LIN {X 0,Y 303.657,Z 547.41,A -85,B 0,C 180,E1 -15927.346,E2 -15927.346} C_VEL
LIN {X 0,Y 303.964,Z 546.683,A -85,B 0,C 180,E1 -15929.999,E2 -15929.999} C_VEL
LIN {X 0,Y 303.831,Z 546.451,A -85,B 0,C 180,E1 -15931.324,E2 -15931.324} C_VEL
LIN {X 0,Y 303.743,Z 545.822,A -85,B 0,C 180,E1 -15932.651,E2 -15932.651} C_VEL
LIN {X 0,Y 303.722,Z 544.801,A -85,B 0,C 180,E1 -15933.979,E2 -15933.979} C_VEL
LIN {X 0,Y 303.711,Z 542.811,A -85,B 0,C 180,E1 -15935.709,E2 -15935.709} C_VEL
LIN {X 0,Y 303.917,Z 539.098,A -85,B 0,C 180,E1 -15937.974,E2 -15937.974} C_VEL
LIN {X 0,Y 304.289,Z 534.652,A -85,B 0,C 180,E1 -15939.974,E2 -15939.974} C_VEL
LIN {X 0,Y 305.086,Z 527.886,A -85,B 0,C 180,E1 -15942.302,E2 -15942.302} C_VEL
LIN {X 0,Y 306.244,Z 520.516,A -85,B 0,C 180,E1 -15944.281,E2 -15944.281} C_VEL
LIN {X 0,Y 307.621,Z 511.711,A -85,B 0,C 180,E1 -15946.178,E2 -15946.178} C_VEL
LIN {X 0,Y 308.984,Z 501.769,A -85,B 0,C 180,E1 -15947.881,E2 -15947.881} C_VEL
LIN {X 0,Y 310.533,Z 491.16,A -85,B 0,C 180,E1 -15949.328,E2 -15949.328} C_VEL
LIN {X 0,Y 311.922,Z 480.889,A -85,B 0,C 180,E1 -15950.439,E2 -15950.439} C_VEL
LIN {X 0,Y 313.304,Z 468.561,A -85,B 0,C 180,E1 -15951.463,E2 -15951.463} C_VEL
LIN {X 0,Y 314.44,Z 455.612,A -85,B 0,C 180,E1 -15952.243,E2 -15952.243} C_VEL
LIN {X 0,Y 315.236,Z 443.183,A -85,B 0,C 180,E1 -15952.731,E2 -15952.731} C_VEL
LIN {X 0,Y 316.694,Z 379.006,A -85,B 0,C 180,E1 -15954.196,E2 -15954.196} C_VEL
LIN {X 0,Y 312.076,Z 344.443,A -85,B 0,C 180,E1 -15955.428,E2 -15955.428} C_VEL
LIN {X 0,Y 309.088,Z 325.843,A -85,B 0,C 180,E1 -15956.169,E2 -15956.169} C_VEL
LIN {X 0,Y 307.11,Z 315.452,A -85,B 0,C 180,E1 -15959.089,E2 -15959.089} C_VEL
LIN {X 0,Y 305.501,Z 307.431,A -85,B 0,C 180,E1 -15961.442,E2 -15961.442} C_VEL
LIN {X 0,Y 305.458,Z 307.433,A -85,B 0,C 180,E1 -15965.112,E2 -15965.112} C_VEL
LIN {X 0,Y 305.462,Z 307.434,A -85,B 0,C 180,E1 -15968.531,E2 -15968.531} C_VEL
LIN {X 0,Y 305.449,Z 307.432,A -85,B 0,C 180,E1 -15972.584,E2 -15972.584} C_VEL
LIN {X 0,Y 305.416,Z 307.436,A -85,B 0,C 180,E1 -15976.343,E2 -15976.343} C_VEL
LIN {X 0,Y 305.403,Z 307.44,A -85,B 0,C 180,E1 -15979.884,E2 -15979.884} C_VEL
LIN {X 0,Y 305.455,Z 307.437,A -85,B 0,C 180,E1 -15983.635,E2 -15983.635} C_VEL
LIN {X 0,Y 305.457,Z 307.433,A -85,B 0,C 180,E1 -15986.482,E2 -15986.482} C_VEL
LIN {X 0,Y 305.41,Z 307.44,A -85,B 0,C 180,E1 -15989.585,E2 -15989.585} C_VEL
LIN {X 0,Y 305.439,Z 307.436,A -85,B 0,C 180,E1 -15992.601,E2 -15992.601} C_VEL
LIN {X 0,Y 305.448,Z 307.436,A -85,B 0,C 180,E1 -15995.534,E2 -15995.534} C_VEL
LIN {X 0,Y 305.475,Z 307.427,A -85,B 0,C 180,E1 -15999.812,E2 -15999.812} C_VEL
LIN {X 0,Y 305.542,Z 307.416,A -85,B 0,C 180,E1 -16003.977,E2 -16003.977} C_VEL
LIN {X 0,Y 305.578,Z 307.417,A -85,B 0,C 180,E1 -16006.703,E2 -16006.703} C_VEL
LIN {X 0,Y 305.744,Z 307.395,A -85,B 0,C 180,E1 -16011.262,E2 -16011.262} C_VEL
LIN {X 0,Y 305.774,Z 307.379,A -85,B 0,C 180,E1 -16013.401,E2 -16013.401} C_VEL
LIN {X 0,Y 305.847,Z 307.383,A -85,B 0,C 180,E1 -16017.366,E2 -16017.366} C_VEL
LIN {X 0,Y 305.903,Z 307.377,A -85,B 0,C 180,E1 -16020,E2 -16020} C_VEL
LIN {X 0,Y 305.842,Z 307.385,A -85,B 0,C 180,E1 -16022.634,E2 -16022.634} C_VEL
LIN {X 0,Y 305.775,Z 307.395,A -85,B 0,C 180,E1 -16026.599,E2 -16026.599} C_VEL
LIN {X 0,Y 305.686,Z 307.404,A -85,B 0,C 180,E1 -16029.261,E2 -16029.261} C_VEL
LIN {X 0,Y 305.578,Z 307.42,A -85,B 0,C 180,E1 -16033.297,E2 -16033.297} C_VEL
LIN {X 0,Y 305.543,Z 307.418,A -85,B 0,C 180,E1 -16036.023,E2 -16036.023} C_VEL
LIN {X 0,Y 305.534,Z 307.424,A -85,B 0,C 180,E1 -16039.427,E2 -16039.427} C_VEL
LIN {X 0,Y 305.479,Z 307.43,A -85,B 0,C 180,E1 -16043.04,E2 -16043.04} C_VEL
LIN {X 0,Y 305.47,Z 307.428,A -85,B 0,C 180,E1 -16046.201,E2 -16046.201} C_VEL
LIN {X 0,Y 305.456,Z 307.435,A -85,B 0,C 180,E1 -16049.04,E2 -16049.04} C_VEL
LIN {X 0,Y 305.43,Z 307.432,A -85,B 0,C 180,E1 -16051.954,E2 -16051.954} C_VEL
LIN {X 0,Y 305.456,Z 307.435,A -85,B 0,C 180,E1 -16055.114,E2 -16055.114} C_VEL
LIN {X 0,Y 305.443,Z 307.435,A -85,B 0,C 180,E1 -16058.53,E2 -16058.53} C_VEL
LIN {X 0,Y 305.449,Z 307.434,A -85,B 0,C 180,E1 -16062.587,E2 -16062.587} C_VEL
LIN {X 0,Y 305.421,Z 307.441,A -85,B 0,C 180,E1 -16066.346,E2 -16066.346} C_VEL
LIN {X 0,Y 305.454,Z 307.436,A -85,B 0,C 180,E1 -16069.894,E2 -16069.894} C_VEL
LIN {X 0,Y 305.478,Z 307.424,A -85,B 0,C 180,E1 -16073.633,E2 -16073.633} C_VEL
LIN {X 0,Y 305.462,Z 307.434,A -85,B 0,C 180,E1 -16076.485,E2 -16076.485} C_VEL
LIN {X 0,Y 305.455,Z 307.433,A -85,B 0,C 180,E1 -16079.592,E2 -16079.592} C_VEL
LIN {X 0,Y 305.526,Z 307.425,A -85,B 0,C 180,E1 -16083.469,E2 -16083.469} C_VEL
LIN {X 0,Y 306.651,Z 310.421,A -85,B 0,C 180,E1 -16083.666,E2 -16083.666} C_VEL
LIN {X 0,Y 315.433,Z 329.159,A -85,B 0,C 180,E1 -16084.926,E2 -16084.926} C_VEL
LIN {X 0,Y 318.099,Z 335.429,A -85,B 0,C 180,E1 -16085.306,E2 -16085.306} C_VEL
LIN {X 0,Y 317.199,Z 379.67,A -85,B 0,C 180,E1 -16086.313,E2 -16086.313} C_VEL
LIN {X 0,Y 316.238,Z 417.455,A -85,B 0,C 180,E1 -16087.201,E2 -16087.201} C_VEL
LIN {X 0,Y 315.569,Z 430.397,A -85,B 0,C 180,E1 -16087.754,E2 -16087.754} C_VEL
LIN {X 0,Y 314.521,Z 443.873,A -85,B 0,C 180,E1 -16088.624,E2 -16088.624} C_VEL
LIN {X 0,Y 313.322,Z 455.582,A -85,B 0,C 180,E1 -16089.656,E2 -16089.656} C_VEL
LIN {X 0,Y 311.905,Z 466.753,A -85,B 0,C 180,E1 -16090.932,E2 -16090.932} C_VEL
LIN {X 0,Y 310.754,Z 476.06,A -85,B 0,C 180,E1 -16092.267,E2 -16092.267} C_VEL
LIN {X 0,Y 309.297,Z 485.106,A -85,B 0,C 180,E1 -16093.84,E2 -16093.84} C_VEL
LIN {X 0,Y 307.998,Z 492.729,A -85,B 0,C 180,E1 -16095.465,E2 -16095.465} C_VEL
LIN {X 0,Y 306.779,Z 500.157,A -85,B 0,C 180,E1 -16097.431,E2 -16097.431} C_VEL
LIN {X 0,Y 305.743,Z 506.122,A -85,B 0,C 180,E1 -16099.405,E2 -16099.405} C_VEL
LIN {X 0,Y 304.994,Z 510.833,A -85,B 0,C 180,E1 -16101.387,E2 -16101.387} C_VEL
LIN {X 0,Y 304.481,Z 514.431,A -85,B 0,C 180,E1 -16103.374,E2 -16103.374} C_VEL
LIN {X 0,Y 304.244,Z 516.283,A -85,B 0,C 180,E1 -16104.7,E2 -16104.7} C_VEL
LIN {X 0,Y 304.001,Z 517.699,A -85,B 0,C 180,E1 -16106.024,E2 -16106.024} C_VEL
LIN {X 0,Y 303.771,Z 519.302,A -85,B 0,C 180,E1 -16108.676,E2 -16108.676} C_VEL
LIN {X 0,Y 303.767,Z 519.534,A -85,B 0,C 180,E1 -16110.001,E2 -16110.001} C_VEL
LIN {X 0,Y 303.771,Z 519.341,A -85,B 0,C 180,E1 -16111.327,E2 -16111.327} C_VEL
LIN {X 0,Y 303.998,Z 517.791,A -85,B 0,C 180,E1 -16113.978,E2 -16113.978} C_VEL
LIN {X 0,Y 304.24,Z 516.425,A -85,B 0,C 180,E1 -16115.303,E2 -16115.303} C_VEL
LIN {X 0,Y 304.624,Z 513.67,A -85,B 0,C 180,E1 -16117.225,E2 -16117.225} C_VEL
LIN {X 0,Y 305.149,Z 509.667,A -85,B 0,C 180,E1 -16119.279,E2 -16119.279} C_VEL
LIN {X 0,Y 306.027,Z 504.616,A -85,B 0,C 180,E1 -16121.258,E2 -16121.258} C_VEL
LIN {X 0,Y 307.119,Z 498.247,A -85,B 0,C 180,E1 -16123.23,E2 -16123.23} C_VEL
LIN {X 0,Y 308.437,Z 490.319,A -85,B 0,C 180,E1 -16125.192,E2 -16125.192} C_VEL
LIN {X 0,Y 309.862,Z 482.199,A -85,B 0,C 180,E1 -16126.81,E2 -16126.81} C_VEL
LIN {X 0,Y 311.249,Z 472.224,A -85,B 0,C 180,E1 -16128.43,E2 -16128.43} C_VEL
LIN {X 0,Y 312.689,Z 461.004,A -85,B 0,C 180,E1 -16129.875,E2 -16129.875} C_VEL
LIN {X 0,Y 313.976,Z 449.96,A -85,B 0,C 180,E1 -16130.987,E2 -16130.987} C_VEL
LIN {X 0,Y 315.116,Z 437.46,A -85,B 0,C 180,E1 -16131.937,E2 -16131.937} C_VEL
LIN {X 0,Y 315.979,Z 424.357,A -85,B 0,C 180,E1 -16132.649,E2 -16132.649} C_VEL
LIN {X 0,Y 316.472,Z 411.322,A -85,B 0,C 180,E1 -16133.086,E2 -16133.086} C_VEL
LIN {X 0,Y 318.254,Z 335.871,A -85,B 0,C 180,E1 -16134.785,E2 -16134.785} C_VEL
LIN {X 0,Y 310.377,Z 318.013,A -85,B 0,C 180,E1 -16135.916,E2 -16135.916} C_VEL
LIN {X 0,Y 305.665,Z 308.157,A -85,B 0,C 180,E1 -16136.604,E2 -16136.604} C_VEL
LIN {X 0,Y 305.53,Z 307.424,A -85,B 0,C 180,E1 -16136.661,E2 -16136.661} C_VEL
LIN {X 0,Y 305.468,Z 307.433,A -85,B 0,C 180,E1 -16140.41,E2 -16140.41} C_VEL
LIN {X 0,Y 305.47,Z 307.434,A -85,B 0,C 180,E1 -16144.079,E2 -16144.079} C_VEL
LIN {X 0,Y 305.501,Z 307.427,A -85,B 0,C 180,E1 -16146.737,E2 -16146.737} C_VEL
LIN {X 0,Y 305.459,Z 307.435,A -85,B 0,C 180,E1 -16150.614,E2 -16150.614} C_VEL
LIN {X 0,Y 305.451,Z 307.432,A -85,B 0,C 180,E1 -16153.652,E2 -16153.652} C_VEL
LIN {X 0,Y 305.448,Z 307.421,A -85,B 0,C 180,E1 -16156.346,E2 -16156.346} C_VEL
LIN {X 0,Y 304.825,Z 307.507,A -85,B 0,C 180,E1 -16157.445,E2 -16157.445} C_VEL
LIN {X 0,Y 301.944,Z 307.873,A -85,B 0,C 180,E1 -16159.235,E2 -16159.235} C_VEL
LIN {X 0,Y 299.493,Z 308.179,A -85,B 0,C 180,E1 -16160.687,E2 -16160.687} C_VEL
LIN {X 0,Y 298.473,Z 308.303,A -85,B 0,C 180,E1 -16161.812,E2 -16161.812} C_VEL
LIN {X 0,Y 298.41,Z 308.31,A -85,B 0,C 180,E1 -16162.194,E2 -16162.194} C_VEL
LIN {X 0,Y 298.414,Z 308.312,A -85,B 0,C 180,E1 -16165.582,E2 -16165.582} C_VEL
LIN {X 0,Y 298.397,Z 308.311,A -85,B 0,C 180,E1 -16168.791,E2 -16168.791} C_VEL
LIN {X 0,Y 298.463,Z 308.305,A -85,B 0,C 180,E1 -16171.904,E2 -16171.904} C_VEL
LIN {X 0,Y 298.52,Z 308.295,A -85,B 0,C 180,E1 -16176.039,E2 -16176.039} C_VEL
LIN {X 0,Y 298.545,Z 308.359,A -85,B 0,C 180,E1 -16176.41,E2 -16176.41} C_VEL
LIN {X 0,Y 298.71,Z 309.327,A -85,B 0,C 180,E1 -16176.684,E2 -16176.684} C_VEL
LIN {X 0,Y 304.792,Z 332.568,A -85,B 0,C 180,E1 -16177.782,E2 -16177.782} C_VEL
LIN {X 0,Y 305.454,Z 337.875,A -85,B 0,C 180,E1 -16177.999,E2 -16177.999} C_VEL
LIN {X 0,Y 302.641,Z 418.79,A -85,B 0,C 180,E1 -16180.852,E2 -16180.852} C_VEL
LIN {X 0,Y 302.093,Z 432.467,A -85,B 0,C 180,E1 -16181.607,E2 -16181.607} C_VEL
LIN {X 0,Y 301.327,Z 444.568,A -85,B 0,C 180,E1 -16182.526,E2 -16182.526} C_VEL
LIN {X 0,Y 300.57,Z 456.641,A -85,B 0,C 180,E1 -16183.705,E2 -16183.705} C_VEL
LIN {X 0,Y 300.027,Z 465.153,A -85,B 0,C 180,E1 -16184.72,E2 -16184.72} C_VEL
LIN {X 0,Y 299.157,Z 475.798,A -85,B 0,C 180,E1 -16186.239,E2 -16186.239} C_VEL
LIN {X 0,Y 298.337,Z 486.282,A -85,B 0,C 180,E1 -16188.104,E2 -16188.104} C_VEL
LIN {X 0,Y 297.698,Z 495.551,A -85,B 0,C 180,E1 -16190.145,E2 -16190.145} C_VEL
LIN {X 0,Y 297.211,Z 502.937,A -85,B 0,C 180,E1 -16192.185,E2 -16192.185} C_VEL
LIN {X 0,Y 296.851,Z 509.748,A -85,B 0,C 180,E1 -16194.566,E2 -16194.566} C_VEL
LIN {X 0,Y 296.772,Z 514.18,A -85,B 0,C 180,E1 -16196.606,E2 -16196.606} C_VEL
LIN {X 0,Y 296.617,Z 517.475,A -85,B 0,C 180,E1 -16198.642,E2 -16198.642} C_VEL
LIN {X 0,Y 296.63,Z 519.071,A -85,B 0,C 180,E1 -16200,E2 -16200} C_VEL
LIN {X 0,Y 296.736,Z 520.242,A -85,B 0,C 180,E1 -16201.357,E2 -16201.357} C_VEL
LIN {X 0,Y 296.924,Z 520.999,A -85,B 0,C 180,E1 -16202.713,E2 -16202.713} C_VEL
LIN {X 0,Y 297.161,Z 521.297,A -85,B 0,C 180,E1 -16204.069,E2 -16204.069} C_VEL
LIN {X 0,Y 297.378,Z 521.168,A -85,B 0,C 180,E1 -16205.424,E2 -16205.424} C_VEL
LIN {X 0,Y 297.751,Z 520.634,A -85,B 0,C 180,E1 -16206.778,E2 -16206.778} C_VEL
LIN {X 0,Y 298.641,Z 519.069,A -85,B 0,C 180,E1 -16208.731,E2 -16208.731} C_VEL
LIN {X 0,Y 300.157,Z 515.318,A -85,B 0,C 180,E1 -16211.48,E2 -16211.48} C_VEL
LIN {X 0,Y 301.698,Z 511.3,A -85,B 0,C 180,E1 -16213.471,E2 -16213.471} C_VEL
LIN {X 0,Y 303.4,Z 506.16,A -85,B 0,C 180,E1 -16215.449,E2 -16215.449} C_VEL
LIN {X 0,Y 305.88,Z 498.522,A -85,B 0,C 180,E1 -16217.724,E2 -16217.724} C_VEL
LIN {X 0,Y 308.402,Z 490.221,A -85,B 0,C 180,E1 -16219.641,E2 -16219.641} C_VEL
LIN {X 0,Y 311.29,Z 479.988,A -85,B 0,C 180,E1 -16221.523,E2 -16221.523} C_VEL
LIN {X 0,Y 314.004,Z 469.151,A -85,B 0,C 180,E1 -16223.104,E2 -16223.104} C_VEL
LIN {X 0,Y 316.565,Z 457.559,A -85,B 0,C 180,E1 -16224.46,E2 -16224.46} C_VEL
LIN {X 0,Y 318.939,Z 444.809,A -85,B 0,C 180,E1 -16225.623,E2 -16225.623} C_VEL
LIN {X 0,Y 320.899,Z 432.294,A -85,B 0,C 180,E1 -16226.502,E2 -16226.502} C_VEL
LIN {X 0,Y 322.631,Z 418.016,A -85,B 0,C 180,E1 -16227.223,E2 -16227.223} C_VEL
LIN {X 0,Y 329.241,Z 360.312,A -85,B 0,C 180,E1 -16229.538,E2 -16229.538} C_VEL
LIN {X 0,Y 325.595,Z 352.92,A -85,B 0,C 180,E1 -16231.008,E2 -16231.008} C_VEL
LIN {X 0,Y 322.312,Z 347.353,A -85,B 0,C 180,E1 -16232.44,E2 -16232.44} C_VEL
LIN {X 0,Y 318.784,Z 341.964,A -85,B 0,C 180,E1 -16234.186,E2 -16234.186} C_VEL
LIN {X 0,Y 315.89,Z 337.946,A -85,B 0,C 180,E1 -16235.88,E2 -16235.88} C_VEL
LIN {X 0,Y 312.534,Z 333.726,A -85,B 0,C 180,E1 -16238.417,E2 -16238.417} C_VEL
LIN {X 0,Y 309.76,Z 331.31,A -85,B 0,C 180,E1 -16241.74,E2 -16241.74} C_VEL
LIN {X 0,Y 309.236,Z 330.576,A -85,B 0,C 180,E1 -16243.341,E2 -16243.341} C_VEL
LIN {X 0,Y 309.074,Z 331.036,A -85,B 0,C 180,E1 -16245.474,E2 -16245.474} C_VEL
LIN {X 0,Y 309.758,Z 332.653,A -85,B 0,C 180,E1 -16247.724,E2 -16247.724} C_VEL
LIN {X 0,Y 311.676,Z 336.685,A -85,B 0,C 180,E1 -16250.482,E2 -16250.482} C_VEL
LIN {X 0,Y 314.583,Z 341.177,A -85,B 0,C 180,E1 -16252.879,E2 -16252.879} C_VEL
LIN {X 0,Y 318.33,Z 348.268,A -85,B 0,C 180,E1 -16255.268,E2 -16255.268} C_VEL
LIN {X 0,Y 321.308,Z 354.437,A -85,B 0,C 180,E1 -16256.849,E2 -16256.849} C_VEL
LIN {X 0,Y 323.815,Z 360.163,A -85,B 0,C 180,E1 -16258.057,E2 -16258.057} C_VEL
LIN {X 0,Y 324.995,Z 363.139,A -85,B 0,C 180,E1 -16258.6,E2 -16258.6} C_VEL
LIN {X 0,Y 326.341,Z 374.009,A -85,B 0,C 180,E1 -16259.718,E2 -16259.718} C_VEL
LIN {X 0,Y 327.059,Z 384.878,A -85,B 0,C 180,E1 -16260.612,E2 -16260.612} C_VEL
LIN {X 0,Y 321.516,Z 436.451,A -85,B 0,C 180,E1 -16262.674,E2 -16262.674} C_VEL
LIN {X 0,Y 319.542,Z 451.172,A -85,B 0,C 180,E1 -16263.375,E2 -16263.375} C_VEL
LIN {X 0,Y 316.795,Z 466.219,A -85,B 0,C 180,E1 -16264.366,E2 -16264.366} C_VEL
LIN {X 0,Y 314.332,Z 477.863,A -85,B 0,C 180,E1 -16265.389,E2 -16265.389} C_VEL
LIN {X 0,Y 311.455,Z 490.024,A -85,B 0,C 180,E1 -16266.74,E2 -16266.74} C_VEL
LIN {X 0,Y 308.656,Z 501.054,A -85,B 0,C 180,E1 -16268.283,E2 -16268.283} C_VEL
LIN {X 0,Y 306.177,Z 510.183,A -85,B 0,C 180,E1 -16269.859,E2 -16269.859} C_VEL
LIN {X 0,Y 303.687,Z 518.633,A -85,B 0,C 180,E1 -16271.619,E2 -16271.619} C_VEL
LIN {X 0,Y 301.519,Z 526.799,A -85,B 0,C 180,E1 -16273.756,E2 -16273.756} C_VEL
LIN {X 0,Y 299.822,Z 532.872,A -85,B 0,C 180,E1 -16275.75,E2 -16275.75} C_VEL
LIN {X 0,Y 298.46,Z 537.761,A -85,B 0,C 180,E1 -16277.763,E2 -16277.763} C_VEL
LIN {X 0,Y 297.5,Z 541.558,A -85,B 0,C 180,E1 -16279.793,E2 -16279.793} C_VEL
LIN {X 0,Y 296.894,Z 544.333,A -85,B 0,C 180,E1 -16281.833,E2 -16281.833} C_VEL
LIN {X 0,Y 296.581,Z 546.422,A -85,B 0,C 180,E1 -16284.422,E2 -16284.422} C_VEL
LIN {X 0,Y 296.572,Z 546.955,A -85,B 0,C 180,E1 -16285.922,E2 -16285.922} C_VEL
LIN {X 0,Y 296.58,Z 546.981,A -85,B 0,C 180,E1 -16287.282,E2 -16287.282} C_VEL
LIN {X 0,Y 296.866,Z 546.366,A -85,B 0,C 180,E1 -16289.999,E2 -16289.999} C_VEL
LIN {X 0,Y 296.735,Z 546.133,A -85,B 0,C 180,E1 -16291.356,E2 -16291.356} C_VEL
LIN {X 0,Y 296.661,Z 545.505,A -85,B 0,C 180,E1 -16292.714,E2 -16292.714} C_VEL
LIN {X 0,Y 296.631,Z 544.483,A -85,B 0,C 180,E1 -16294.075,E2 -16294.075} C_VEL
LIN {X 0,Y 296.623,Z 542.739,A -85,B 0,C 180,E1 -16295.659,E2 -16295.659} C_VEL
LIN {X 0,Y 296.852,Z 538.78,A -85,B 0,C 180,E1 -16298.165,E2 -16298.165} C_VEL
LIN {X 0,Y 297.251,Z 534.333,A -85,B 0,C 180,E1 -16300.213,E2 -16300.213} C_VEL
LIN {X 0,Y 297.94,Z 528.667,A -85,B 0,C 180,E1 -16302.256,E2 -16302.256} C_VEL
LIN {X 0,Y 299.15,Z 521.553,A -85,B 0,C 180,E1 -16304.28,E2 -16304.28} C_VEL
LIN {X 0,Y 300.572,Z 512.685,A -85,B 0,C 180,E1 -16306.294,E2 -16306.294} C_VEL
LIN {X 0,Y 301.899,Z 503.565,A -85,B 0,C 180,E1 -16307.964,E2 -16307.964} C_VEL
LIN {X 0,Y 303.457,Z 493.414,A -85,B 0,C 180,E1 -16309.445,E2 -16309.445} C_VEL
LIN {X 0,Y 305.071,Z 482.154,A -85,B 0,C 180,E1 -16310.743,E2 -16310.743} C_VEL
LIN {X 0,Y 306.465,Z 470.457,A -85,B 0,C 180,E1 -16311.789,E2 -16311.789} C_VEL
LIN {X 0,Y 307.691,Z 457.555,A -85,B 0,C 180,E1 -16312.625,E2 -16312.625} C_VEL
LIN {X 0,Y 308.64,Z 444.389,A -85,B 0,C 180,E1 -16313.193,E2 -16313.193} C_VEL
LIN {X 0,Y 309.973,Z 393.218,A -85,B 0,C 180,E1 -16314.397,E2 -16314.397} C_VEL
LIN {X 0,Y 310.199,Z 379.909,A -85,B 0,C 180,E1 -16314.708,E2 -16314.708} C_VEL
LIN {X 0,Y 305.808,Z 346.318,A -85,B 0,C 180,E1 -16315.934,E2 -16315.934} C_VEL
LIN {X 0,Y 302.785,Z 328.078,A -85,B 0,C 180,E1 -16316.681,E2 -16316.681} C_VEL
LIN {X 0,Y 301.693,Z 324.321,A -85,B 0,C 180,E1 -16316.9,E2 -16316.9} C_VEL
LIN {X 0,Y 298.974,Z 310.991,A -85,B 0,C 180,E1 -16320.779,E2 -16320.779} C_VEL
LIN {X 0,Y 298.462,Z 308.308,A -85,B 0,C 180,E1 -16321.635,E2 -16321.635} C_VEL
LIN {X 0,Y 298.415,Z 308.314,A -85,B 0,C 180,E1 -16326.068,E2 -16326.068} C_VEL
LIN {X 0,Y 298.404,Z 308.313,A -85,B 0,C 180,E1 -16329.485,E2 -16329.485} C_VEL
LIN {X 0,Y 298.394,Z 308.311,A -85,B 0,C 180,E1 -16333.102,E2 -16333.102} C_VEL
LIN {X 0,Y 298.365,Z 308.312,A -85,B 0,C 180,E1 -16336.914,E2 -16336.914} C_VEL
LIN {X 0,Y 298.344,Z 308.314,A -85,B 0,C 180,E1 -16341.018,E2 -16341.018} C_VEL
LIN {X 0,Y 298.397,Z 308.312,A -85,B 0,C 180,E1 -16343.927,E2 -16343.927} C_VEL
LIN {X 0,Y 298.385,Z 308.315,A -85,B 0,C 180,E1 -16347.198,E2 -16347.198} C_VEL
LIN {X 0,Y 298.36,Z 308.316,A -85,B 0,C 180,E1 -16350.636,E2 -16350.636} C_VEL
LIN {X 0,Y 298.413,Z 308.308,A -85,B 0,C 180,E1 -16354.917,E2 -16354.917} C_VEL
LIN {X 0,Y 298.393,Z 308.315,A -85,B 0,C 180,E1 -16357.862,E2 -16357.862} C_VEL
LIN {X 0,Y 298.456,Z 308.299,A -85,B 0,C 180,E1 -16360.751,E2 -16360.751} C_VEL
LIN {X 0,Y 298.578,Z 308.283,A -85,B 0,C 180,E1 -16364.994,E2 -16364.994} C_VEL
LIN {X 0,Y 298.574,Z 308.294,A -85,B 0,C 180,E1 -16369.146,E2 -16369.146} C_VEL
LIN {X 0,Y 298.687,Z 308.268,A -85,B 0,C 180,E1 -16371.884,E2 -16371.884} C_VEL
LIN {X 0,Y 298.619,Z 308.264,A -85,B 0,C 180,E1 -16374.598,E2 -16374.598} C_VEL
LIN {X 0,Y 298.894,Z 308.249,A -85,B 0,C 180,E1 -16378.653,E2 -16378.653} C_VEL
LIN {X 0,Y 298.903,Z 308.251,A -85,B 0,C 180,E1 -16381.347,E2 -16381.347} C_VEL
LIN {X 0,Y 298.724,Z 308.275,A -85,B 0,C 180,E1 -16386.756,E2 -16386.756} C_VEL
LIN {X 0,Y 298.617,Z 308.282,A -85,B 0,C 180,E1 -16389.483,E2 -16389.483} C_VEL
LIN {X 0,Y 298.537,Z 308.295,A -85,B 0,C 180,E1 -16393.616,E2 -16393.616} C_VEL
LIN {X 0,Y 298.478,Z 308.299,A -85,B 0,C 180,E1 -16396.413,E2 -16396.413} C_VEL
LIN {X 0,Y 298.475,Z 308.302,A -85,B 0,C 180,E1 -16399.64,E2 -16399.64} C_VEL
LIN {X 0,Y 298.417,Z 308.306,A -85,B 0,C 180,E1 -16403.601,E2 -16403.601} C_VEL
LIN {X 0,Y 298.409,Z 308.31,A -85,B 0,C 180,E1 -16406.582,E2 -16406.582} C_VEL
LIN {X 0,Y 298.393,Z 308.313,A -85,B 0,C 180,E1 -16409.644,E2 -16409.644} C_VEL
LIN {X 0,Y 298.386,Z 308.313,A -85,B 0,C 180,E1 -16412.802,E2 -16412.802} C_VEL
LIN {X 0,Y 298.44,Z 308.306,A -85,B 0,C 180,E1 -16416.809,E2 -16416.809} C_VEL
LIN {X 0,Y 298.381,Z 308.315,A -85,B 0,C 180,E1 -16421.089,E2 -16421.089} C_VEL
LIN {X 0,Y 298.393,Z 308.311,A -85,B 0,C 180,E1 -16423.105,E2 -16423.105} C_VEL
LIN {X 0,Y 298.398,Z 308.311,A -85,B 0,C 180,E1 -16426.922,E2 -16426.922} C_VEL
LIN {X 0,Y 298.411,Z 308.308,A -85,B 0,C 180,E1 -16431.005,E2 -16431.005} C_VEL
LIN {X 0,Y 298.415,Z 308.305,A -85,B 0,C 180,E1 -16433.932,E2 -16433.932} C_VEL
LIN {X 0,Y 298.39,Z 308.309,A -85,B 0,C 180,E1 -16437.985,E2 -16437.985} C_VEL
LIN {X 0,Y 298.457,Z 308.307,A -85,B 0,C 180,E1 -16441.905,E2 -16441.905} C_VEL
LIN {X 0,Y 298.479,Z 308.303,A -85,B 0,C 180,E1 -16442.811,E2 -16442.811} C_VEL
LIN {X 0,Y 299.494,Z 311.154,A -85,B 0,C 180,E1 -16442.999,E2 -16442.999} C_VEL
LIN {X 0,Y 307.474,Z 327.59,A -85,B 0,C 180,E1 -16444.183,E2 -16444.183} C_VEL
LIN {X 0,Y 311.683,Z 337.348,A -85,B 0,C 180,E1 -16444.805,E2 -16444.805} C_VEL
LIN {X 0,Y 309.917,Z 412.201,A -85,B 0,C 180,E1 -16446.532,E2 -16446.532} C_VEL
LIN {X 0,Y 309.396,Z 424.986,A -85,B 0,C 180,E1 -16446.977,E2 -16446.977} C_VEL
LIN {X 0,Y 308.563,Z 437.395,A -85,B 0,C 180,E1 -16447.663,E2 -16447.663} C_VEL
LIN {X 0,Y 307.42,Z 449.046,A -85,B 0,C 180,E1 -16448.546,E2 -16448.546} C_VEL
LIN {X 0,Y 306.108,Z 460.416,A -85,B 0,C 180,E1 -16449.682,E2 -16449.682} C_VEL
LIN {X 0,Y 304.604,Z 471.8,A -85,B 0,C 180,E1 -16451.156,E2 -16451.156} C_VEL
LIN {X 0,Y 303.114,Z 481.944,A -85,B 0,C 180,E1 -16452.807,E2 -16452.807} C_VEL
LIN {X 0,Y 301.637,Z 490.16,A -85,B 0,C 180,E1 -16454.46,E2 -16454.46} C_VEL
LIN {X 0,Y 300.276,Z 498.161,A -85,B 0,C 180,E1 -16456.466,E2 -16456.466} C_VEL
LIN {X 0,Y 299.123,Z 504.606,A -85,B 0,C 180,E1 -16458.481,E2 -16458.481} C_VEL
LIN {X 0,Y 298.209,Z 509.728,A -85,B 0,C 180,E1 -16460.506,E2 -16460.506} C_VEL
LIN {X 0,Y 297.56,Z 514.026,A -85,B 0,C 180,E1 -16462.744,E2 -16462.744} C_VEL
LIN {X 0,Y 297.178,Z 516.6,A -85,B 0,C 180,E1 -16464.573,E2 -16464.573} C_VEL
LIN {X 0,Y 296.941,Z 518.015,A -85,B 0,C 180,E1 -16465.93,E2 -16465.93} C_VEL
LIN {X 0,Y 296.684,Z 519.619,A -85,B 0,C 180,E1 -16468.644,E2 -16468.644} C_VEL
LIN {X 0,Y 296.675,Z 519.851,A -85,B 0,C 180,E1 -16470.001,E2 -16470.001} C_VEL
LIN {X 0,Y 296.684,Z 519.658,A -85,B 0,C 180,E1 -16471.359,E2 -16471.359} C_VEL
LIN {X 0,Y 296.938,Z 518.106,A -85,B 0,C 180,E1 -16474.073,E2 -16474.073} C_VEL
LIN {X 0,Y 297.174,Z 516.741,A -85,B 0,C 180,E1 -16475.43,E2 -16475.43} C_VEL
LIN {X 0,Y 297.542,Z 514.242,A -85,B 0,C 180,E1 -16477.229,E2 -16477.229} C_VEL
LIN {X 0,Y 298.132,Z 509.982,A -85,B 0,C 180,E1 -16479.499,E2 -16479.499} C_VEL
LIN {X 0,Y 299.074,Z 504.929,A -85,B 0,C 180,E1 -16481.523,E2 -16481.523} C_VEL
LIN {X 0,Y 300.229,Z 498.558,A -85,B 0,C 180,E1 -16483.539,E2 -16483.539} C_VEL
LIN {X 0,Y 301.595,Z 490.629,A -85,B 0,C 180,E1 -16485.545,E2 -16485.545} C_VEL
LIN {X 0,Y 303.068,Z 482.507,A -85,B 0,C 180,E1 -16487.199,E2 -16487.199} C_VEL
LIN {X 0,Y 304.525,Z 472.528,A -85,B 0,C 180,E1 -16488.852,E2 -16488.852} C_VEL
LIN {X 0,Y 306.038,Z 461.303,A -85,B 0,C 180,E1 -16490.326,E2 -16490.326} C_VEL
LIN {X 0,Y 307.389,Z 450.25,A -85,B 0,C 180,E1 -16491.459,E2 -16491.459} C_VEL
LIN {X 0,Y 308.549,Z 437.738,A -85,B 0,C 180,E1 -16492.429,E2 -16492.429} C_VEL
LIN {X 0,Y 309.467,Z 424.613,A -85,B 0,C 180,E1 -16493.153,E2 -16493.153} C_VEL
LIN {X 0,Y 309.978,Z 411.518,A -85,B 0,C 180,E1 -16493.599,E2 -16493.599} C_VEL
LIN {X 0,Y 311.805,Z 337.588,A -85,B 0,C 180,E1 -16495.295,E2 -16495.295} C_VEL
LIN {X 0,Y 303.699,Z 319.52,A -85,B 0,C 180,E1 -16496.495,E2 -16496.495} C_VEL
LIN {X 0,Y 298.704,Z 309.41,A -85,B 0,C 180,E1 -16497.246,E2 -16497.246} C_VEL
LIN {X 0,Y 298.483,Z 308.303,A -85,B 0,C 180,E1 -16497.337,E2 -16497.337} C_VEL
LIN {X 0,Y 298.401,Z 308.315,A -85,B 0,C 180,E1 -16501.21,E2 -16501.21} C_VEL
LIN {X 0,Y 298.433,Z 308.309,A -85,B 0,C 180,E1 -16504.488,E2 -16504.488} C_VEL
LIN {X 0,Y 298.437,Z 308.314,A -85,B 0,C 180,E1 -16507.756,E2 -16507.756} C_VEL
LIN {X 0,Y 298.418,Z 308.316,A -85,B 0,C 180,E1 -16511.257,E2 -16511.257} C_VEL
LIN {X 0,Y 298.394,Z 308.302,A -85,B 0,C 180,E1 -16515.042,E2 -16515.042} C_VEL
LIN {X 0,Y 298.393,Z 308.312,A -85,B 0,C 180,E1 -16518.913,E2 -16518.913} C_VEL
LIN {X 0,Y 298.41,Z 308.31,A -85,B 0,C 180,E1 -16522.194,E2 -16522.194} C_VEL
LIN {X 0,Y 297.805,Z 308.388,A -85,B 0,C 180,E1 -16523.32,E2 -16523.32} C_VEL
LIN {X 0,Y 294.995,Z 308.742,A -85,B 0,C 180,E1 -16525.155,E2 -16525.155} C_VEL
LIN {X 0,Y 292.552,Z 309.045,A -85,B 0,C 180,E1 -16526.643,E2 -16526.643} C_VEL
LIN {X 0,Y 291.464,Z 309.175,A -85,B 0,C 180,E1 -16527.796,E2 -16527.796} C_VEL
LIN {X 0,Y 291.356,Z 309.186,A -85,B 0,C 180,E1 -16528.187,E2 -16528.187} C_VEL
LIN {X 0,Y 291.383,Z 309.19,A -85,B 0,C 180,E1 -16531.158,E2 -16531.158} C_VEL
LIN {X 0,Y 291.424,Z 309.182,A -85,B 0,C 180,E1 -16534.272,E2 -16534.272} C_VEL
LIN {X 0,Y 291.506,Z 309.237,A -85,B 0,C 180,E1 -16536.296,E2 -16536.296} C_VEL
LIN {X 0,Y 291.676,Z 310.186,A -85,B 0,C 180,E1 -16536.419,E2 -16536.419} C_VEL
LIN {X 0,Y 297.96,Z 334.104,A -85,B 0,C 180,E1 -16537.575,E2 -16537.575} C_VEL
LIN {X 0,Y 298.474,Z 338.793,A -85,B 0,C 180,E1 -16537.769,E2 -16537.769} C_VEL
LIN {X 0,Y 295.601,Z 418.979,A -85,B 0,C 180,E1 -16540.693,E2 -16540.693} C_VEL
LIN {X 0,Y 295.063,Z 431.929,A -85,B 0,C 180,E1 -16541.423,E2 -16541.423} C_VEL
LIN {X 0,Y 294.265,Z 444.694,A -85,B 0,C 180,E1 -16542.406,E2 -16542.406} C_VEL
LIN {X 0,Y 293.495,Z 457.182,A -85,B 0,C 180,E1 -16543.658,E2 -16543.658} C_VEL
LIN {X 0,Y 292.742,Z 466.921,A -85,B 0,C 180,E1 -16544.866,E2 -16544.866} C_VEL
LIN {X 0,Y 291.98,Z 477.288,A -85,B 0,C 180,E1 -16546.427,E2 -16546.427} C_VEL
LIN {X 0,Y 291.239,Z 486.725,A -85,B 0,C 180,E1 -16548.164,E2 -16548.164} C_VEL
LIN {X 0,Y 290.585,Z 495.975,A -85,B 0,C 180,E1 -16550.253,E2 -16550.253} C_VEL
LIN {X 0,Y 290.104,Z 503.347,A -85,B 0,C 180,E1 -16552.343,E2 -16552.343} C_VEL
LIN {X 0,Y 289.762,Z 509.262,A -85,B 0,C 180,E1 -16554.432,E2 -16554.432} C_VEL
LIN {X 0,Y 289.703,Z 513.907,A -85,B 0,C 180,E1 -16556.523,E2 -16556.523} C_VEL
LIN {X 0,Y 289.535,Z 517.377,A -85,B 0,C 180,E1 -16558.609,E2 -16558.609} C_VEL
LIN {X 0,Y 289.543,Z 519.13,A -85,B 0,C 180,E1 -16560,E2 -16560} C_VEL
LIN {X 0,Y 289.651,Z 520.395,A -85,B 0,C 180,E1 -16561.39,E2 -16561.39} C_VEL
LIN {X 0,Y 289.845,Z 521.241,A -85,B 0,C 180,E1 -16562.78,E2 -16562.78} C_VEL
LIN {X 0,Y 290.093,Z 521.68,A -85,B 0,C 180,E1 -16564.168,E2 -16564.168} C_VEL
LIN {X 0,Y 290.338,Z 521.682,A -85,B 0,C 180,E1 -16565.556,E2 -16565.556} C_VEL
LIN {X 0,Y 290.746,Z 521.239,A -85,B 0,C 180,E1 -16566.942,E2 -16566.942} C_VEL
LIN {X 0,Y 291.628,Z 519.953,A -85,B 0,C 180,E1 -16568.854,E2 -16568.854} C_VEL
LIN {X 0,Y 292.867,Z 517.396,A -85,B 0,C 180,E1 -16571.068,E2 -16571.068} C_VEL
LIN {X 0,Y 294.321,Z 513.971,A -85,B 0,C 180,E1 -16573.112,E2 -16573.112} C_VEL
LIN {X 0,Y 296.097,Z 509.454,A -85,B 0,C 180,E1 -16575.135,E2 -16575.135} C_VEL
LIN {X 0,Y 298.551,Z 502.662,A -85,B 0,C 180,E1 -16577.466,E2 -16577.466} C_VEL
LIN {X 0,Y 301.052,Z 495.315,A -85,B 0,C 180,E1 -16579.431,E2 -16579.431} C_VEL
LIN {X 0,Y 304.011,Z 486.192,A -85,B 0,C 180,E1 -16581.352,E2 -16581.352} C_VEL
LIN {X 0,Y 306.678,Z 476.998,A -85,B 0,C 180,E1 -16582.928,E2 -16582.928} C_VEL
LIN {X 0,Y 309.672,Z 465.282,A -85,B 0,C 180,E1 -16584.537,E2 -16584.537} C_VEL
LIN {X 0,Y 312.406,Z 453.335,A -85,B 0,C 180,E1 -16585.827,E2 -16585.827} C_VEL
LIN {X 0,Y 314.905,Z 439.905,A -85,B 0,C 180,E1 -16586.958,E2 -16586.958} C_VEL
LIN {X 0,Y 316.949,Z 426.354,A -85,B 0,C 180,E1 -16587.797,E2 -16587.797} C_VEL
LIN {X 0,Y 319.915,Z 401.675,A -85,B 0,C 180,E1 -16588.857,E2 -16588.857} C_VEL
LIN {X 0,Y 324.727,Z 363.654,A -85,B 0,C 180,E1 -16590.418,E2 -16590.418} C_VEL
LIN {X 0,Y 321.115,Z 356.412,A -85,B 0,C 180,E1 -16592.015,E2 -16592.015} C_VEL
LIN {X 0,Y 317.892,Z 351.072,A -85,B 0,C 180,E1 -16593.584,E2 -16593.584} C_VEL
LIN {X 0,Y 315.809,Z 347.805,A -85,B 0,C 180,E1 -16594.738,E2 -16594.738} C_VEL
LIN {X 0,Y 313.516,Z 344.415,A -85,B 0,C 180,E1 -16596.194,E2 -16596.194} C_VEL
LIN {X 0,Y 310.458,Z 340.42,A -85,B 0,C 180,E1 -16598.649,E2 -16598.649} C_VEL
LIN {X 0,Y 307.94,Z 338.163,A -85,B 0,C 180,E1 -16601.805,E2 -16601.805} C_VEL
LIN {X 0,Y 307.483,Z 337.449,A -85,B 0,C 180,E1 -16603.291,E2 -16603.291} C_VEL
LIN {X 0,Y 307.309,Z 337.933,A -85,B 0,C 180,E1 -16605.501,E2 -16605.501} C_VEL
LIN {X 0,Y 307.856,Z 339.382,A -85,B 0,C 180,E1 -16607.506,E2 -16607.506} C_VEL
LIN {X 0,Y 309.649,Z 343.454,A -85,B 0,C 180,E1 -16610.305,E2 -16610.305} C_VEL
LIN {X 0,Y 312.102,Z 347.41,A -85,B 0,C 180,E1 -16612.453,E2 -16612.453} C_VEL
LIN {X 0,Y 315.442,Z 354.239,A -85,B 0,C 180,E1 -16614.793,E2 -16614.793} C_VEL
LIN {X 0,Y 318.162,Z 360.205,A -85,B 0,C 180,E1 -16616.358,E2 -16616.358} C_VEL
LIN {X 0,Y 320.276,Z 365.358,A -85,B 0,C 180,E1 -16617.471,E2 -16617.471} C_VEL
LIN {X 0,Y 321.118,Z 367.772,A -85,B 0,C 180,E1 -16617.907,E2 -16617.907} C_VEL
LIN {X 0,Y 322.129,Z 378.466,A -85,B 0,C 180,E1 -16619.006,E2 -16619.006} C_VEL
LIN {X 0,Y 322.536,Z 387.202,A -85,B 0,C 180,E1 -16619.736,E2 -16619.736} C_VEL
LIN {X 0,Y 315.689,Z 444.125,A -85,B 0,C 180,E1 -16622.081,E2 -16622.081} C_VEL
LIN {X 0,Y 313.28,Z 458.11,A -85,B 0,C 180,E1 -16622.89,E2 -16622.89} C_VEL
LIN {X 0,Y 310.646,Z 470.479,A -85,B 0,C 180,E1 -16623.821,E2 -16623.821} C_VEL
LIN {X 0,Y 307.816,Z 482.536,A -85,B 0,C 180,E1 -16625.013,E2 -16625.013} C_VEL
LIN {X 0,Y 304.514,Z 494.826,A -85,B 0,C 180,E1 -16626.538,E2 -16626.538} C_VEL
LIN {X 0,Y 301.713,Z 504.862,A -85,B 0,C 180,E1 -16628.117,E2 -16628.117} C_VEL
LIN {X 0,Y 298.711,Z 514.812,A -85,B 0,C 180,E1 -16630.052,E2 -16630.052} C_VEL
LIN {X 0,Y 296.048,Z 523.013,A -85,B 0,C 180,E1 -16632.023,E2 -16632.023} C_VEL
LIN {X 0,Y 294.117,Z 529.673,A -85,B 0,C 180,E1 -16634.049,E2 -16634.049} C_VEL
LIN {X 0,Y 292.341,Z 535.103,A -85,B 0,C 180,E1 -16636.088,E2 -16636.088} C_VEL
LIN {X 0,Y 291.145,Z 539.395,A -85,B 0,C 180,E1 -16638.158,E2 -16638.158} C_VEL
LIN {X 0,Y 290.268,Z 542.659,A -85,B 0,C 180,E1 -16640.241,E2 -16640.241} C_VEL
LIN {X 0,Y 289.587,Z 545.453,A -85,B 0,C 180,E1 -16643.029,E2 -16643.029} C_VEL
LIN {X 0,Y 289.482,Z 546.276,A -85,B 0,C 180,E1 -16644.5,E2 -16644.5} C_VEL
LIN {X 0,Y 289.488,Z 546.589,A -85,B 0,C 180,E1 -16645.822,E2 -16645.822} C_VEL
LIN {X 0,Y 289.504,Z 546.482,A -85,B 0,C 180,E1 -16647.216,E2 -16647.216} C_VEL
LIN {X 0,Y 289.58,Z 545.957,A -85,B 0,C 180,E1 -16648.608,E2 -16648.608} C_VEL
LIN {X 0,Y 289.769,Z 546.049,A -85,B 0,C 180,E1 -16649.999,E2 -16649.999} C_VEL
LIN {X 0,Y 289.643,Z 545.816,A -85,B 0,C 180,E1 -16651.389,E2 -16651.389} C_VEL
LIN {X 0,Y 289.581,Z 545.188,A -85,B 0,C 180,E1 -16652.781,E2 -16652.781} C_VEL
LIN {X 0,Y 289.525,Z 544.165,A -85,B 0,C 180,E1 -16654.175,E2 -16654.175} C_VEL
LIN {X 0,Y 289.516,Z 542.715,A -85,B 0,C 180,E1 -16655.571,E2 -16655.571} C_VEL
LIN {X 0,Y 289.701,Z 539.711,A -85,B 0,C 180,E1 -16657.666,E2 -16657.666} C_VEL
LIN {X 0,Y 290.049,Z 535.638,A -85,B 0,C 180,E1 -16659.764,E2 -16659.764} C_VEL
LIN {X 0,Y 290.826,Z 529.362,A -85,B 0,C 180,E1 -16662.206,E2 -16662.206} C_VEL
LIN {X 0,Y 292.031,Z 522.536,A -85,B 0,C 180,E1 -16664.279,E2 -16664.279} C_VEL
LIN {X 0,Y 293.208,Z 515.561,A -85,B 0,C 180,E1 -16665.999,E2 -16665.999} C_VEL
LIN {X 0,Y 294.509,Z 507.137,A -85,B 0,C 180,E1 -16667.712,E2 -16667.712} C_VEL
LIN {X 0,Y 296.144,Z 496.707,A -85,B 0,C 180,E1 -16669.403,E2 -16669.403} C_VEL
LIN {X 0,Y 297.784,Z 486.389,A -85,B 0,C 180,E1 -16670.731,E2 -16670.731} C_VEL
LIN {X 0,Y 299.297,Z 475.051,A -85,B 0,C 180,E1 -16671.885,E2 -16671.885} C_VEL
LIN {X 0,Y 300.725,Z 462.054,A -85,B 0,C 180,E1 -16672.861,E2 -16672.861} C_VEL
LIN {X 0,Y 301.808,Z 449.314,A -85,B 0,C 180,E1 -16673.529,E2 -16673.529} C_VEL
LIN {X 0,Y 302.458,Z 436.44,A -85,B 0,C 180,E1 -16673.938,E2 -16673.938} C_VEL
LIN {X 0,Y 303.708,Z 380.371,A -85,B 0,C 180,E1 -16675.255,E2 -16675.255} C_VEL
LIN {X 0,Y 299.502,Z 347.889,A -85,B 0,C 180,E1 -16676.476,E2 -16676.476} C_VEL
LIN {X 0,Y 296.676,Z 330.559,A -85,B 0,C 180,E1 -16677.204,E2 -16677.204} C_VEL
LIN {X 0,Y 294.128,Z 322.688,A -85,B 0,C 180,E1 -16677.692,E2 -16677.692} C_VEL
LIN {X 0,Y 291.44,Z 309.182,A -85,B 0,C 180,E1 -16681.785,E2 -16681.785} C_VEL
LIN {X 0,Y 291.358,Z 309.191,A -85,B 0,C 180,E1 -16685.372,E2 -16685.372} C_VEL
LIN {X 0,Y 291.359,Z 309.19,A -85,B 0,C 180,E1 -16688.839,E2 -16688.839} C_VEL
LIN {X 0,Y 291.314,Z 309.193,A -85,B 0,C 180,E1 -16692.491,E2 -16692.491} C_VEL
LIN {X 0,Y 291.283,Z 309.195,A -85,B 0,C 180,E1 -16696.369,E2 -16696.369} C_VEL
LIN {X 0,Y 291.304,Z 309.191,A -85,B 0,C 180,E1 -16700.534,E2 -16700.534} C_VEL
LIN {X 0,Y 291.379,Z 309.186,A -85,B 0,C 180,E1 -16702.915,E2 -16702.915} C_VEL
LIN {X 0,Y 291.336,Z 309.192,A -85,B 0,C 180,E1 -16706.3,E2 -16706.3} C_VEL
LIN {X 0,Y 291.329,Z 309.193,A -85,B 0,C 180,E1 -16710.277,E2 -16710.277} C_VEL
LIN {X 0,Y 291.338,Z 309.188,A -85,B 0,C 180,E1 -16714.264,E2 -16714.264} C_VEL
LIN {X 0,Y 291.351,Z 309.194,A -85,B 0,C 180,E1 -16717.297,E2 -16717.297} C_VEL
LIN {X 0,Y 291.384,Z 309.179,A -85,B 0,C 180,E1 -16720.265,E2 -16720.265} C_VEL
LIN {X 0,Y 291.489,Z 309.164,A -85,B 0,C 180,E1 -16724.665,E2 -16724.665} C_VEL
LIN {X 0,Y 291.52,Z 309.171,A -85,B 0,C 180,E1 -16728.88,E2 -16728.88} C_VEL
LIN {X 0,Y 291.641,Z 309.145,A -85,B 0,C 180,E1 -16731.687,E2 -16731.687} C_VEL
LIN {X 0,Y 291.588,Z 309.138,A -85,B 0,C 180,E1 -16734.468,E2 -16734.468} C_VEL
LIN {X 0,Y 291.862,Z 309.124,A -85,B 0,C 180,E1 -16738.62,E2 -16738.62} C_VEL
LIN {X 0,Y 291.869,Z 309.126,A -85,B 0,C 180,E1 -16741.38,E2 -16741.38} C_VEL
LIN {X 0,Y 291.676,Z 309.154,A -85,B 0,C 180,E1 -16746.92,E2 -16746.92} C_VEL
LIN {X 0,Y 291.559,Z 309.16,A -85,B 0,C 180,E1 -16749.714,E2 -16749.714} C_VEL
LIN {X 0,Y 291.507,Z 309.171,A -85,B 0,C 180,E1 -16753.951,E2 -16753.951} C_VEL
LIN {X 0,Y 291.425,Z 309.175,A -85,B 0,C 180,E1 -16756.822,E2 -16756.822} C_VEL
LIN {X 0,Y 291.416,Z 309.182,A -85,B 0,C 180,E1 -16759.861,E2 -16759.861} C_VEL
LIN {X 0,Y 291.359,Z 309.186,A -85,B 0,C 180,E1 -16764.209,E2 -16764.209} C_VEL
LIN {X 0,Y 291.355,Z 309.191,A -85,B 0,C 180,E1 -16767.279,E2 -16767.279} C_VEL
LIN {X 0,Y 291.315,Z 309.196,A -85,B 0,C 180,E1 -16770.44,E2 -16770.44} C_VEL
LIN {X 0,Y 291.337,Z 309.191,A -85,B 0,C 180,E1 -16773.7,E2 -16773.7} C_VEL
LIN {X 0,Y 291.37,Z 309.184,A -85,B 0,C 180,E1 -16777.255,E2 -16777.255} C_VEL
LIN {X 0,Y 291.327,Z 309.197,A -85,B 0,C 180,E1 -16780.644,E2 -16780.644} C_VEL
LIN {X 0,Y 291.285,Z 309.2,A -85,B 0,C 180,E1 -16784.403,E2 -16784.403} C_VEL
LIN {X 0,Y 291.322,Z 309.196,A -85,B 0,C 180,E1 -16788.406,E2 -16788.406} C_VEL
LIN {X 0,Y 291.36,Z 309.186,A -85,B 0,C 180,E1 -16791.161,E2 -16791.161} C_VEL
LIN {X 0,Y 291.358,Z 309.191,A -85,B 0,C 180,E1 -16794.628,E2 -16794.628} C_VEL
LIN {X 0,Y 291.367,Z 309.183,A -85,B 0,C 180,E1 -16797.952,E2 -16797.952} C_VEL
LIN {X 0,Y 291.452,Z 309.332,A -85,B 0,C 180,E1 -16802.133,E2 -16802.133} C_VEL
LIN {X 0,Y 292.537,Z 312.17,A -85,B 0,C 180,E1 -16802.324,E2 -16802.324} C_VEL
LIN {X 0,Y 300.979,Z 329.394,A -85,B 0,C 180,E1 -16803.624,E2 -16803.624} C_VEL
LIN {X 0,Y 305.268,Z 339.223,A -85,B 0,C 180,E1 -16804.28,E2 -16804.28} C_VEL
LIN {X 0,Y 303.269,Z 416.655,A -85,B 0,C 180,E1 -16806.122,E2 -16806.122} C_VEL
LIN {X 0,Y 302.637,Z 429.478,A -85,B 0,C 180,E1 -16806.659,E2 -16806.659} C_VEL
LIN {X 0,Y 301.569,Z 442.327,A -85,B 0,C 180,E1 -16807.478,E2 -16807.478} C_VEL
LIN {X 0,Y 300.268,Z 454.568,A -85,B 0,C 180,E1 -16808.55,E2 -16808.55} C_VEL
LIN {X 0,Y 298.885,Z 464.85,A -85,B 0,C 180,E1 -16809.708,E2 -16809.708} C_VEL
LIN {X 0,Y 297.44,Z 475.665,A -85,B 0,C 180,E1 -16811.27,E2 -16811.27} C_VEL
LIN {X 0,Y 295.717,Z 485.733,A -85,B 0,C 180,E1 -16813.076,E2 -16813.076} C_VEL
LIN {X 0,Y 294.261,Z 493.361,A -85,B 0,C 180,E1 -16814.77,E2 -16814.77} C_VEL
LIN {X 0,Y 292.962,Z 500.789,A -85,B 0,C 180,E1 -16816.828,E2 -16816.828} C_VEL
LIN {X 0,Y 291.81,Z 506.755,A -85,B 0,C 180,E1 -16818.893,E2 -16818.893} C_VEL
LIN {X 0,Y 290.977,Z 511.467,A -85,B 0,C 180,E1 -16820.969,E2 -16820.969} C_VEL
LIN {X 0,Y 290.411,Z 515.064,A -85,B 0,C 180,E1 -16823.052,E2 -16823.052} C_VEL
LIN {X 0,Y 290.116,Z 516.917,A -85,B 0,C 180,E1 -16824.441,E2 -16824.441} C_VEL
LIN {X 0,Y 289.882,Z 518.332,A -85,B 0,C 180,E1 -16825.83,E2 -16825.83} C_VEL
LIN {X 0,Y 289.599,Z 519.936,A -85,B 0,C 180,E1 -16828.611,E2 -16828.611} C_VEL
LIN {X 0,Y 289.587,Z 520.167,A -85,B 0,C 180,E1 -16830.001,E2 -16830.001} C_VEL
LIN {X 0,Y 289.599,Z 519.974,A -85,B 0,C 180,E1 -16831.392,E2 -16831.392} C_VEL
LIN {X 0,Y 289.879,Z 518.421,A -85,B 0,C 180,E1 -16834.172,E2 -16834.172} C_VEL
LIN {X 0,Y 290.112,Z 517.057,A -85,B 0,C 180,E1 -16835.562,E2 -16835.562} C_VEL
LIN {X 0,Y 290.481,Z 514.768,A -85,B 0,C 180,E1 -16837.264,E2 -16837.264} C_VEL
LIN {X 0,Y 291.138,Z 510.297,A -85,B 0,C 180,E1 -16839.73,E2 -16839.73} C_VEL
LIN {X 0,Y 292.131,Z 505.242,A -85,B 0,C 180,E1 -16841.801,E2 -16841.801} C_VEL
LIN {X 0,Y 293.327,Z 498.871,A -85,B 0,C 180,E1 -16843.864,E2 -16843.864} C_VEL
LIN {X 0,Y 294.756,Z 490.939,A -85,B 0,C 180,E1 -16845.916,E2 -16845.916} C_VEL
LIN {X 0,Y 296.302,Z 482.815,A -85,B 0,C 180,E1 -16847.604,E2 -16847.604} C_VEL
LIN {X 0,Y 297.826,Z 472.831,A -85,B 0,C 180,E1 -16849.292,E2 -16849.292} C_VEL
LIN {X 0,Y 299.409,Z 461.601,A -85,B 0,C 180,E1 -16850.796,E2 -16850.796} C_VEL
LIN {X 0,Y 300.818,Z 450.54,A -85,B 0,C 180,E1 -16851.952,E2 -16851.952} C_VEL
LIN {X 0,Y 302.02,Z 438.017,A -85,B 0,C 180,E1 -16852.942,E2 -16852.942} C_VEL
LIN {X 0,Y 302.902,Z 425.717,A -85,B 0,C 180,E1 -16853.64,E2 -16853.64} C_VEL
LIN {X 0,Y 303.488,Z 413.317,A -85,B 0,C 180,E1 -16854.09,E2 -16854.09} C_VEL
LIN {X 0,Y 305.366,Z 339.421,A -85,B 0,C 180,E1 -16855.825,E2 -16855.825} C_VEL
LIN {X 0,Y 296.999,Z 320.914,A -85,B 0,C 180,E1 -16857.109,E2 -16857.109} C_VEL
LIN {X 0,Y 291.643,Z 310.187,A -85,B 0,C 180,E1 -16857.947,E2 -16857.947} C_VEL
LIN {X 0,Y 291.443,Z 309.179,A -85,B 0,C 180,E1 -16858.024,E2 -16858.024} C_VEL
LIN {X 0,Y 291.35,Z 309.193,A -85,B 0,C 180,E1 -16862.405,E2 -16862.405} C_VEL
LIN {X 0,Y 291.39,Z 309.19,A -85,B 0,C 180,E1 -16865.371,E2 -16865.371} C_VEL
LIN {X 0,Y 291.37,Z 309.192,A -85,B 0,C 180,E1 -16868.84,E2 -16868.84} C_VEL
LIN {X 0,Y 291.353,Z 309.193,A -85,B 0,C 180,E1 -16872.488,E2 -16872.488} C_VEL
LIN {X 0,Y 291.324,Z 309.177,A -85,B 0,C 180,E1 -16876.365,E2 -16876.365} C_VEL
LIN {X 0,Y 291.384,Z 309.188,A -85,B 0,C 180,E1 -16880.519,E2 -16880.519} C_VEL
LIN {X 0,Y 291.409,Z 309.182,A -85,B 0,C 180,E1 -16882.92,E2 -16882.92} C_VEL
LIN {X 0,Y 291.35,Z 309.192,A -85,B 0,C 180,E1 -16886.302,E2 -16886.302} C_VEL
LIN {X 0,Y 291.356,Z 309.186,A -85,B 0,C 180,E1 -16888.187,E2 -16888.187} C_VEL
LIN {X 0,Y 290.645,Z 309.275,A -85,B 0,C 180,E1 -16889.341,E2 -16889.341} C_VEL
LIN {X 0,Y 287.81,Z 309.634,A -85,B 0,C 180,E1 -16891.222,E2 -16891.222} C_VEL
LIN {X 0,Y 285.443,Z 309.931,A -85,B 0,C 180,E1 -16892.749,E2 -16892.749} C_VEL
LIN {X 0,Y 284.438,Z 310.051,A -85,B 0,C 180,E1 -16893.931,E2 -16893.931} C_VEL
LIN {X 0,Y 284.36,Z 310.056,A -85,B 0,C 180,E1 -16894.332,E2 -16894.332} C_VEL
LIN {X 0,Y 284.438,Z 310.069,A -85,B 0,C 180,E1 -16896.097,E2 -16896.097} C_VEL
LIN {X 0,Y 291.189,Z 335.97,A -85,B 0,C 180,E1 -16897.383,E2 -16897.383} C_VEL
LIN {X 0,Y 291.46,Z 339.727,A -85,B 0,C 180,E1 -16897.538,E2 -16897.538} C_VEL
LIN {X 0,Y 288.572,Z 418.814,A -85,B 0,C 180,E1 -16900.528,E2 -16900.528} C_VEL
LIN {X 0,Y 287.983,Z 432.505,A -85,B 0,C 180,E1 -16901.318,E2 -16901.318} C_VEL
LIN {X 0,Y 287.15,Z 445.866,A -85,B 0,C 180,E1 -16902.388,E2 -16902.388} C_VEL
LIN {X 0,Y 286.4,Z 457.907,A -85,B 0,C 180,E1 -16903.642,E2 -16903.642} C_VEL
LIN {X 0,Y 285.489,Z 468.56,A -85,B 0,C 180,E1 -16905.02,E2 -16905.02} C_VEL
LIN {X 0,Y 284.783,Z 478.667,A -85,B 0,C 180,E1 -16906.623,E2 -16906.623} C_VEL
LIN {X 0,Y 283.988,Z 488.792,A -85,B 0,C 180,E1 -16908.581,E2 -16908.581} C_VEL
LIN {X 0,Y 283.381,Z 497.662,A -85,B 0,C 180,E1 -16910.723,E2 -16910.723} C_VEL
LIN {X 0,Y 282.914,Z 504.802,A -85,B 0,C 180,E1 -16912.865,E2 -16912.865} C_VEL
LIN {X 0,Y 282.639,Z 510.511,A -85,B 0,C 180,E1 -16915.007,E2 -16915.007} C_VEL
LIN {X 0,Y 282.561,Z 514.951,A -85,B 0,C 180,E1 -16917.149,E2 -16917.149} C_VEL
LIN {X 0,Y 282.455,Z 517.248,A -85,B 0,C 180,E1 -16918.574,E2 -16918.574} C_VEL
LIN {X 0,Y 282.459,Z 519.099,A -85,B 0,C 180,E1 -16920,E2 -16920} C_VEL
LIN {X 0,Y 282.568,Z 520.526,A -85,B 0,C 180,E1 -16921.425,E2 -16921.425} C_VEL
LIN {X 0,Y 282.77,Z 521.477,A -85,B 0,C 180,E1 -16922.849,E2 -16922.849} C_VEL
LIN {X 0,Y 283.028,Z 522.01,A -85,B 0,C 180,E1 -16924.272,E2 -16924.272} C_VEL
LIN {X 0,Y 283.302,Z 522.143,A -85,B 0,C 180,E1 -16925.695,E2 -16925.695} C_VEL
LIN {X 0,Y 283.746,Z 521.853,A -85,B 0,C 180,E1 -16927.114,E2 -16927.114} C_VEL
LIN {X 0,Y 284.619,Z 520.778,A -85,B 0,C 180,E1 -16928.987,E2 -16928.987} C_VEL
LIN {X 0,Y 285.974,Z 518.39,A -85,B 0,C 180,E1 -16931.338,E2 -16931.338} C_VEL
LIN {X 0,Y 287.533,Z 515.182,A -85,B 0,C 180,E1 -16933.427,E2 -16933.427} C_VEL
LIN {X 0,Y 289.412,Z 510.915,A -85,B 0,C 180,E1 -16935.493,E2 -16935.493} C_VEL
LIN {X 0,Y 292.014,Z 504.439,A -85,B 0,C 180,E1 -16937.87,E2 -16937.87} C_VEL
LIN {X 0,Y 294.639,Z 497.433,A -85,B 0,C 180,E1 -16939.871,E2 -16939.871} C_VEL
LIN {X 0,Y 297.744,Z 488.809,A -85,B 0,C 180,E1 -16941.825,E2 -16941.825} C_VEL
LIN {X 0,Y 300.544,Z 480.058,A -85,B 0,C 180,E1 -16943.424,E2 -16943.424} C_VEL
LIN {X 0,Y 303.905,Z 468.355,A -85,B 0,C 180,E1 -16945.147,E2 -16945.147} C_VEL
LIN {X 0,Y 306.882,Z 456.403,A -85,B 0,C 180,E1 -16946.524,E2 -16946.524} C_VEL
LIN {X 0,Y 309.674,Z 443.103,A -85,B 0,C 180,E1 -16947.725,E2 -16947.725} C_VEL
LIN {X 0,Y 311.945,Z 430.051,A -85,B 0,C 180,E1 -16948.604,E2 -16948.604} C_VEL
LIN {X 0,Y 313.862,Z 415.713,A -85,B 0,C 180,E1 -16949.302,E2 -16949.302} C_VEL
LIN {X 0,Y 320.329,Z 367.05,A -85,B 0,C 180,E1 -16951.354,E2 -16951.354} C_VEL
LIN {X 0,Y 317.269,Z 360.929,A -85,B 0,C 180,E1 -16952.842,E2 -16952.842} C_VEL
LIN {X 0,Y 314.732,Z 356.597,A -85,B 0,C 180,E1 -16954.2,E2 -16954.2} C_VEL
LIN {X 0,Y 313.137,Z 353.982,A -85,B 0,C 180,E1 -16955.16,E2 -16955.16} C_VEL
LIN {X 0,Y 311.059,Z 350.789,A -85,B 0,C 180,E1 -16956.58,E2 -16956.58} C_VEL
LIN {X 0,Y 308.423,Z 347.159,A -85,B 0,C 180,E1 -16958.848,E2 -16958.848} C_VEL
LIN {X 0,Y 306.044,Z 344.884,A -85,B 0,C 180,E1 -16962.084,E2 -16962.084} C_VEL
LIN {X 0,Y 305.627,Z 344.302,A -85,B 0,C 180,E1 -16963.619,E2 -16963.619} C_VEL
LIN {X 0,Y 305.636,Z 345.179,A -85,B 0,C 180,E1 -16966.133,E2 -16966.133} C_VEL
LIN {X 0,Y 306.139,Z 346.657,A -85,B 0,C 180,E1 -16967.733,E2 -16967.733} C_VEL
LIN {X 0,Y 308.14,Z 351.11,A -85,B 0,C 180,E1 -16970.659,E2 -16970.659} C_VEL
LIN {X 0,Y 309.735,Z 353.928,A -85,B 0,C 180,E1 -16972.118,E2 -16972.118} C_VEL
LIN {X 0,Y 312.674,Z 360.3,A -85,B 0,C 180,E1 -16974.337,E2 -16974.337} C_VEL
LIN {X 0,Y 315.043,Z 365.99,A -85,B 0,C 180,E1 -16975.845,E2 -16975.845} C_VEL
LIN {X 0,Y 317.101,Z 371.292,A -85,B 0,C 180,E1 -16977.014,E2 -16977.014} C_VEL
LIN {X 0,Y 317.834,Z 378.497,A -85,B 0,C 180,E1 -16977.846,E2 -16977.846} C_VEL
LIN {X 0,Y 318.193,Z 388.304,A -85,B 0,C 180,E1 -16978.727,E2 -16978.727} C_VEL
LIN {X 0,Y 311.073,Z 443.637,A -85,B 0,C 180,E1 -16981.076,E2 -16981.076} C_VEL
LIN {X 0,Y 308.766,Z 456.428,A -85,B 0,C 180,E1 -16981.815,E2 -16981.815} C_VEL
LIN {X 0,Y 305.347,Z 471.408,A -85,B 0,C 180,E1 -16982.961,E2 -16982.961} C_VEL
LIN {X 0,Y 302.004,Z 484.397,A -85,B 0,C 180,E1 -16984.314,E2 -16984.314} C_VEL
LIN {X 0,Y 298.548,Z 496.161,A -85,B 0,C 180,E1 -16985.856,E2 -16985.856} C_VEL
LIN {X 0,Y 295.302,Z 506.73,A -85,B 0,C 180,E1 -16987.616,E2 -16987.616} C_VEL
LIN {X 0,Y 292.177,Z 516.216,A -85,B 0,C 180,E1 -16989.586,E2 -16989.586} C_VEL
LIN {X 0,Y 289.387,Z 524.017,A -85,B 0,C 180,E1 -16991.595,E2 -16991.595} C_VEL
LIN {X 0,Y 287.346,Z 530.387,A -85,B 0,C 180,E1 -16993.663,E2 -16993.663} C_VEL
LIN {X 0,Y 285.475,Z 535.573,A -85,B 0,C 180,E1 -16995.747,E2 -16995.747} C_VEL
LIN {X 0,Y 284.2,Z 539.641,A -85,B 0,C 180,E1 -16997.865,E2 -16997.865} C_VEL
LIN {X 0,Y 283.236,Z 542.696,A -85,B 0,C 180,E1 -16999.996,E2 -16999.996} C_VEL
LIN {X 0,Y 282.807,Z 544.202,A -85,B 0,C 180,E1 -17001.424,E2 -17001.424} C_VEL
LIN {X 0,Y 282.511,Z 545.296,A -85,B 0,C 180,E1 -17002.853,E2 -17002.853} C_VEL
LIN {X 0,Y 282.384,Z 546.012,A -85,B 0,C 180,E1 -17004.579,E2 -17004.579} C_VEL
LIN {X 0,Y 282.431,Z 545.975,A -85,B 0,C 180,E1 -17007.146,E2 -17007.146} C_VEL
LIN {X 0,Y 282.493,Z 545.507,A -85,B 0,C 180,E1 -17008.573,E2 -17008.573} C_VEL
LIN {X 0,Y 282.671,Z 545.732,A -85,B 0,C 180,E1 -17009.999,E2 -17009.999} C_VEL
LIN {X 0,Y 282.553,Z 545.499,A -85,B 0,C 180,E1 -17011.424,E2 -17011.424} C_VEL
LIN {X 0,Y 282.501,Z 544.872,A -85,B 0,C 180,E1 -17012.851,E2 -17012.851} C_VEL
LIN {X 0,Y 282.422,Z 542.639,A -85,B 0,C 180,E1 -17015.501,E2 -17015.501} C_VEL
LIN {X 0,Y 282.631,Z 539.392,A -85,B 0,C 180,E1 -17017.859,E2 -17017.859} C_VEL
LIN {X 0,Y 283.024,Z 535.319,A -85,B 0,C 180,E1 -17020.009,E2 -17020.009} C_VEL
LIN {X 0,Y 283.838,Z 529.044,A -85,B 0,C 180,E1 -17022.511,E2 -17022.511} C_VEL
LIN {X 0,Y 285.103,Z 522.218,A -85,B 0,C 180,E1 -17024.634,E2 -17024.634} C_VEL
LIN {X 0,Y 286.535,Z 514.149,A -85,B 0,C 180,E1 -17026.642,E2 -17026.642} C_VEL
LIN {X 0,Y 288.024,Z 504.883,A -85,B 0,C 180,E1 -17028.493,E2 -17028.493} C_VEL
LIN {X 0,Y 289.649,Z 495.23,A -85,B 0,C 180,E1 -17030.041,E2 -17030.041} C_VEL
LIN {X 0,Y 291.364,Z 484.657,A -85,B 0,C 180,E1 -17031.396,E2 -17031.396} C_VEL
LIN {X 0,Y 292.919,Z 472.8,A -85,B 0,C 180,E1 -17032.573,E2 -17032.573} C_VEL
LIN {X 0,Y 294.341,Z 460.487,A -85,B 0,C 180,E1 -17033.48,E2 -17033.48} C_VEL
LIN {X 0,Y 295.393,Z 448.279,A -85,B 0,C 180,E1 -17034.109,E2 -17034.109} C_VEL
LIN {X 0,Y 296.057,Z 433.632,A -85,B 0,C 180,E1 -17034.558,E2 -17034.558} C_VEL
LIN {X 0,Y 297.301,Z 381.311,A -85,B 0,C 180,E1 -17035.809,E2 -17035.809} C_VEL
LIN {X 0,Y 293.214,Z 349.351,A -85,B 0,C 180,E1 -17037.044,E2 -17037.044} C_VEL
LIN {X 0,Y 290.67,Z 333.157,A -85,B 0,C 180,E1 -17037.738,E2 -17037.738} C_VEL
LIN {X 0,Y 286.579,Z 321.024,A -85,B 0,C 180,E1 -17038.529,E2 -17038.529} C_VEL
LIN {X 0,Y 284.374,Z 310.062,A -85,B 0,C 180,E1 -17041.938,E2 -17041.938} C_VEL
LIN {X 0,Y 284.33,Z 310.065,A -85,B 0,C 180,E1 -17046.384,E2 -17046.384} C_VEL
LIN {X 0,Y 284.302,Z 310.069,A -85,B 0,C 180,E1 -17049.993,E2 -17049.993} C_VEL
LIN {X 0,Y 284.241,Z 310.077,A -85,B 0,C 180,E1 -17054.189,E2 -17054.189} C_VEL
LIN {X 0,Y 284.234,Z 310.078,A -85,B 0,C 180,E1 -17058.117,E2 -17058.117} C_VEL
LIN {X 0,Y 284.275,Z 310.072,A -85,B 0,C 180,E1 -17062.288,E2 -17062.288} C_VEL
LIN {X 0,Y 284.3,Z 310.066,A -85,B 0,C 180,E1 -17065.349,E2 -17065.349} C_VEL
LIN {X 0,Y 284.271,Z 310.071,A -85,B 0,C 180,E1 -17068.723,E2 -17068.723} C_VEL
LIN {X 0,Y 284.255,Z 310.077,A -85,B 0,C 180,E1 -17071.981,E2 -17071.981} C_VEL
LIN {X 0,Y 284.302,Z 310.069,A -85,B 0,C 180,E1 -17076.151,E2 -17076.151} C_VEL
LIN {X 0,Y 284.326,Z 310.059,A -85,B 0,C 180,E1 -17079.927,E2 -17079.927} C_VEL
LIN {X 0,Y 284.438,Z 310.041,A -85,B 0,C 180,E1 -17084.493,E2 -17084.493} C_VEL
LIN {X 0,Y 284.474,Z 310.047,A -85,B 0,C 180,E1 -17088.601,E2 -17088.601} C_VEL
LIN {X 0,Y 284.598,Z 310.023,A -85,B 0,C 180,E1 -17091.479,E2 -17091.479} C_VEL
LIN {X 0,Y 284.558,Z 310.011,A -85,B 0,C 180,E1 -17094.33,E2 -17094.33} C_VEL
LIN {X 0,Y 284.829,Z 310,A -85,B 0,C 180,E1 -17098.586,E2 -17098.586} C_VEL
LIN {X 0,Y 284.835,Z 310.002,A -85,B 0,C 180,E1 -17101.414,E2 -17101.414} C_VEL
LIN {X 0,Y 284.632,Z 310.031,A -85,B 0,C 180,E1 -17107.092,E2 -17107.092} C_VEL
LIN {X 0,Y 284.506,Z 310.038,A -85,B 0,C 180,E1 -17109.958,E2 -17109.958} C_VEL
LIN {X 0,Y 284.455,Z 310.05,A -85,B 0,C 180,E1 -17114.304,E2 -17114.304} C_VEL
LIN {X 0,Y 284.354,Z 310.059,A -85,B 0,C 180,E1 -17118.742,E2 -17118.742} C_VEL
LIN {X 0,Y 284.307,Z 310.068,A -85,B 0,C 180,E1 -17121.765,E2 -17121.765} C_VEL
LIN {X 0,Y 284.308,Z 310.062,A -85,B 0,C 180,E1 -17124.85,E2 -17124.85} C_VEL
LIN {X 0,Y 284.284,Z 310.071,A -85,B 0,C 180,E1 -17128.016,E2 -17128.016} C_VEL
LIN {X 0,Y 284.28,Z 310.065,A -85,B 0,C 180,E1 -17131.276,E2 -17131.276} C_VEL
LIN {X 0,Y 284.335,Z 310.065,A -85,B 0,C 180,E1 -17135.349,E2 -17135.349} C_VEL
LIN {X 0,Y 284.306,Z 310.064,A -85,B 0,C 180,E1 -17138.17,E2 -17138.17} C_VEL
LIN {X 0,Y 284.264,Z 310.075,A -85,B 0,C 180,E1 -17142.126,E2 -17142.126} C_VEL
LIN {X 0,Y 284.251,Z 310.079,A -85,B 0,C 180,E1 -17146.191,E2 -17146.191} C_VEL
LIN {X 0,Y 284.303,Z 310.072,A -85,B 0,C 180,E1 -17150.025,E2 -17150.025} C_VEL
LIN {X 0,Y 284.331,Z 310.056,A -85,B 0,C 180,E1 -17153.616,E2 -17153.616} C_VEL
LIN {X 0,Y 284.304,Z 310.065,A -85,B 0,C 180,E1 -17157.191,E2 -17157.191} C_VEL
LIN {X 0,Y 284.347,Z 310.063,A -85,B 0,C 180,E1 -17161.359,E2 -17161.359} C_VEL
LIN {X 0,Y 285.421,Z 313.001,A -85,B 0,C 180,E1 -17161.588,E2 -17161.588} C_VEL
LIN {X 0,Y 293.15,Z 328.247,A -85,B 0,C 180,E1 -17162.824,E2 -17162.824} C_VEL
LIN {X 0,Y 298.824,Z 340.999,A -85,B 0,C 180,E1 -17163.724,E2 -17163.724} C_VEL
LIN {X 0,Y 297.834,Z 380.59,A -85,B 0,C 180,E1 -17164.675,E2 -17164.675} C_VEL
LIN {X 0,Y 296.769,Z 418.229,A -85,B 0,C 180,E1 -17165.611,E2 -17165.611} C_VEL
LIN {X 0,Y 295.995,Z 431.264,A -85,B 0,C 180,E1 -17166.196,E2 -17166.196} C_VEL
LIN {X 0,Y 294.843,Z 444.771,A -85,B 0,C 180,E1 -17167.12,E2 -17167.12} C_VEL
LIN {X 0,Y 293.504,Z 456.499,A -85,B 0,C 180,E1 -17168.215,E2 -17168.215} C_VEL
LIN {X 0,Y 291.871,Z 467.678,A -85,B 0,C 180,E1 -17169.566,E2 -17169.566} C_VEL
LIN {X 0,Y 290.471,Z 477.661,A -85,B 0,C 180,E1 -17171.101,E2 -17171.101} C_VEL
LIN {X 0,Y 288.945,Z 486.047,A -85,B 0,C 180,E1 -17172.667,E2 -17172.667} C_VEL
LIN {X 0,Y 287.414,Z 493.676,A -85,B 0,C 180,E1 -17174.398,E2 -17174.398} C_VEL
LIN {X 0,Y 286.044,Z 501.105,A -85,B 0,C 180,E1 -17176.504,E2 -17176.504} C_VEL
LIN {X 0,Y 284.854,Z 507.072,A -85,B 0,C 180,E1 -17178.618,E2 -17178.618} C_VEL
LIN {X 0,Y 283.967,Z 511.784,A -85,B 0,C 180,E1 -17180.744,E2 -17180.744} C_VEL
LIN {X 0,Y 283.357,Z 515.382,A -85,B 0,C 180,E1 -17182.878,E2 -17182.878} C_VEL
LIN {X 0,Y 283.059,Z 517.234,A -85,B 0,C 180,E1 -17184.302,E2 -17184.302} C_VEL
LIN {X 0,Y 282.825,Z 518.648,A -85,B 0,C 180,E1 -17185.726,E2 -17185.726} C_VEL
LIN {X 0,Y 282.517,Z 520.252,A -85,B 0,C 180,E1 -17188.576,E2 -17188.576} C_VEL
LIN {X 0,Y 282.501,Z 520.484,A -85,B 0,C 180,E1 -17190.001,E2 -17190.001} C_VEL
LIN {X 0,Y 282.517,Z 520.29,A -85,B 0,C 180,E1 -17191.427,E2 -17191.427} C_VEL
LIN {X 0,Y 282.823,Z 518.737,A -85,B 0,C 180,E1 -17194.277,E2 -17194.277} C_VEL
LIN {X 0,Y 283.055,Z 517.373,A -85,B 0,C 180,E1 -17195.701,E2 -17195.701} C_VEL
LIN {X 0,Y 283.517,Z 514.508,A -85,B 0,C 180,E1 -17197.837,E2 -17197.837} C_VEL
LIN {X 0,Y 284.163,Z 510.61,A -85,B 0,C 180,E1 -17199.971,E2 -17199.971} C_VEL
LIN {X 0,Y 285.198,Z 505.555,A -85,B 0,C 180,E1 -17202.092,E2 -17202.092} C_VEL
LIN {X 0,Y 286.447,Z 499.182,A -85,B 0,C 180,E1 -17204.204,E2 -17204.204} C_VEL
LIN {X 0,Y 287.947,Z 491.249,A -85,B 0,C 180,E1 -17206.302,E2 -17206.302} C_VEL
LIN {X 0,Y 289.557,Z 483.122,A -85,B 0,C 180,E1 -17208.028,E2 -17208.028} C_VEL
LIN {X 0,Y 291.148,Z 473.134,A -85,B 0,C 180,E1 -17209.753,E2 -17209.753} C_VEL
LIN {X 0,Y 292.787,Z 461.9,A -85,B 0,C 180,E1 -17211.289,E2 -17211.289} C_VEL
LIN {X 0,Y 294.272,Z 450.831,A -85,B 0,C 180,E1 -17212.467,E2 -17212.467} C_VEL
LIN {X 0,Y 295.516,Z 438.295,A -85,B 0,C 180,E1 -17213.476,E2 -17213.476} C_VEL
LIN {X 0,Y 296.44,Z 425.976,A -85,B 0,C 180,E1 -17214.188,E2 -17214.188} C_VEL
LIN {X 0,Y 297.04,Z 413.515,A -85,B 0,C 180,E1 -17214.647,E2 -17214.647} C_VEL
LIN {X 0,Y 298.87,Z 341.076,A -85,B 0,C 180,E1 -17216.39,E2 -17216.39} C_VEL
LIN {X 0,Y 290.333,Z 322.375,A -85,B 0,C 180,E1 -17217.749,E2 -17217.749} C_VEL
LIN {X 0,Y 284.559,Z 311.094,A -85,B 0,C 180,E1 -17218.686,E2 -17218.686} C_VEL
LIN {X 0,Y 284.351,Z 310.063,A -85,B 0,C 180,E1 -17218.778,E2 -17218.778} C_VEL
LIN {X 0,Y 284.311,Z 310.07,A -85,B 0,C 180,E1 -17222.946,E2 -17222.946} C_VEL
LIN {X 0,Y 284.355,Z 310.062,A -85,B 0,C 180,E1 -17226.384,E2 -17226.384} C_VEL
LIN {X 0,Y 284.317,Z 310.07,A -85,B 0,C 180,E1 -17229.994,E2 -17229.994} C_VEL
LIN {X 0,Y 284.282,Z 310.065,A -85,B 0,C 180,E1 -17234.198,E2 -17234.198} C_VEL
LIN {X 0,Y 284.278,Z 310.067,A -85,B 0,C 180,E1 -17238.125,E2 -17238.125} C_VEL
LIN {X 0,Y 284.324,Z 310.065,A -85,B 0,C 180,E1 -17242.279,E2 -17242.279} C_VEL
LIN {X 0,Y 284.314,Z 310.07,A -85,B 0,C 180,E1 -17245.351,E2 -17245.351} C_VEL
LIN {X 0,Y 284.299,Z 310.066,A -85,B 0,C 180,E1 -17248.726,E2 -17248.726} C_VEL
LIN {X 0,Y 284.4,Z 310.061,A -85,B 0,C 180,E1 -17252.828,E2 -17252.828} C_VEL
LIN {X 0,Y 284.36,Z 310.056,A -85,B 0,C 180,E1 -17254.332,E2 -17254.332} C_VEL
LIN {X 0,Y 284.323,Z 310.658,A -85,B 0,C 180,E1 -17254.86,E2 -17254.86} C_VEL
LIN {X 0,Y 284.203,Z 312.741,A -85,B 0,C 180,E1 -17255.465,E2 -17255.465} C_VEL
LIN {X 0,Y 284.004,Z 316.581,A -85,B 0,C 180,E1 -17256.048,E2 -17256.048} C_VEL
LIN {X 0,Y 283.834,Z 322.288,A -85,B 0,C 180,E1 -17256.509,E2 -17256.509} C_VEL
LIN {X 0,Y 284.355,Z 337.729,A -85,B 0,C 180,E1 -17257.191,E2 -17257.191} C_VEL
LIN {X 0,Y 283.979,Z 355.068,A -85,B 0,C 180,E1 -17257.872,E2 -17257.872} C_VEL
LIN {X 0,Y 281.499,Z 419.286,A -85,B 0,C 180,E1 -17260.398,E2 -17260.398} C_VEL
LIN {X 0,Y 280.892,Z 432.838,A -85,B 0,C 180,E1 -17261.208,E2 -17261.208} C_VEL
LIN {X 0,Y 280.089,Z 445.961,A -85,B 0,C 180,E1 -17262.287,E2 -17262.287} C_VEL
LIN {X 0,Y 279.322,Z 458.443,A -85,B 0,C 180,E1 -17263.619,E2 -17263.619} C_VEL
LIN {X 0,Y 278.367,Z 470.086,A -85,B 0,C 180,E1 -17265.189,E2 -17265.189} C_VEL
LIN {X 0,Y 277.557,Z 479.964,A -85,B 0,C 180,E1 -17266.827,E2 -17266.827} C_VEL
LIN {X 0,Y 276.881,Z 489.084,A -85,B 0,C 180,E1 -17268.655,E2 -17268.655} C_VEL
LIN {X 0,Y 276.241,Z 497.953,A -85,B 0,C 180,E1 -17270.85,E2 -17270.85} C_VEL
LIN {X 0,Y 275.791,Z 505.233,A -85,B 0,C 180,E1 -17273.084,E2 -17273.084} C_VEL
LIN {X 0,Y 275.563,Z 511.647,A -85,B 0,C 180,E1 -17275.612,E2 -17275.612} C_VEL
LIN {X 0,Y 275.414,Z 515.894,A -85,B 0,C 180,E1 -17277.806,E2 -17277.806} C_VEL
LIN {X 0,Y 275.377,Z 519.041,A -85,B 0,C 180,E1 -17280,E2 -17280} C_VEL
LIN {X 0,Y 275.488,Z 520.565,A -85,B 0,C 180,E1 -17281.462,E2 -17281.462} C_VEL
LIN {X 0,Y 275.696,Z 521.679,A -85,B 0,C 180,E1 -17282.922,E2 -17282.922} C_VEL
LIN {X 0,Y 275.968,Z 522.338,A -85,B 0,C 180,E1 -17284.382,E2 -17284.382} C_VEL
LIN {X 0,Y 276.271,Z 522.571,A -85,B 0,C 180,E1 -17285.84,E2 -17285.84} C_VEL
LIN {X 0,Y 276.725,Z 522.402,A -85,B 0,C 180,E1 -17287.295,E2 -17287.295} C_VEL
LIN {X 0,Y 277.566,Z 521.62,A -85,B 0,C 180,E1 -17289.068,E2 -17289.068} C_VEL
LIN {X 0,Y 279.088,Z 519.35,A -85,B 0,C 180,E1 -17291.622,E2 -17291.622} C_VEL
LIN {X 0,Y 280.743,Z 516.378,A -85,B 0,C 180,E1 -17293.758,E2 -17293.758} C_VEL
LIN {X 0,Y 282.738,Z 512.358,A -85,B 0,C 180,E1 -17295.868,E2 -17295.868} C_VEL
LIN {X 0,Y 285.073,Z 507.207,A -85,B 0,C 180,E1 -17297.949,E2 -17297.949} C_VEL
LIN {X 0,Y 287.74,Z 500.817,A -85,B 0,C 180,E1 -17299.996,E2 -17299.996} C_VEL
LIN {X 0,Y 290.945,Z 492.897,A -85,B 0,C 180,E1 -17301.988,E2 -17301.988} C_VEL
LIN {X 0,Y 294.436,Z 483.129,A -85,B 0,C 180,E1 -17303.94,E2 -17303.94} C_VEL
LIN {X 0,Y 297.51,Z 473.599,A -85,B 0,C 180,E1 -17305.476,E2 -17305.476} C_VEL
LIN {X 0,Y 300.69,Z 462.441,A -85,B 0,C 180,E1 -17306.927,E2 -17306.927} C_VEL
LIN {X 0,Y 303.614,Z 450.709,A -85,B 0,C 180,E1 -17308.141,E2 -17308.141} C_VEL
LIN {X 0,Y 306.274,Z 437.727,A -85,B 0,C 180,E1 -17309.184,E2 -17309.184} C_VEL
LIN {X 0,Y 308.659,Z 423.57,A -85,B 0,C 180,E1 -17310.014,E2 -17310.014} C_VEL
LIN {X 0,Y 316.164,Z 370.786,A -85,B 0,C 180,E1 -17312.295,E2 -17312.295} C_VEL
LIN {X 0,Y 313.601,Z 365.572,A -85,B 0,C 180,E1 -17313.683,E2 -17313.683} C_VEL
LIN {X 0,Y 310.68,Z 360.422,A -85,B 0,C 180,E1 -17315.473,E2 -17315.473} C_VEL
LIN {X 0,Y 308.697,Z 357.244,A -85,B 0,C 180,E1 -17316.919,E2 -17316.919} C_VEL
LIN {X 0,Y 306.431,Z 353.928,A -85,B 0,C 180,E1 -17318.996,E2 -17318.996} C_VEL
LIN {X 0,Y 304.175,Z 351.633,A -85,B 0,C 180,E1 -17322.321,E2 -17322.321} C_VEL
LIN {X 0,Y 303.793,Z 351.22,A -85,B 0,C 180,E1 -17323.95,E2 -17323.95} C_VEL
LIN {X 0,Y 303.923,Z 352.294,A -85,B 0,C 180,E1 -17326.47,E2 -17326.47} C_VEL
LIN {X 0,Y 304.884,Z 355.292,A -85,B 0,C 180,E1 -17328.88,E2 -17328.88} C_VEL
LIN {X 0,Y 307.253,Z 359.999,A -85,B 0,C 180,E1 -17331.615,E2 -17331.615} C_VEL
LIN {X 0,Y 309.844,Z 366.171,A -85,B 0,C 180,E1 -17333.811,E2 -17333.811} C_VEL
LIN {X 0,Y 311.885,Z 371.38,A -85,B 0,C 180,E1 -17335.236,E2 -17335.236} C_VEL
LIN {X 0,Y 313.57,Z 376.148,A -85,B 0,C 180,E1 -17336.313,E2 -17336.313} C_VEL
LIN {X 0,Y 314.049,Z 385.976,A -85,B 0,C 180,E1 -17337.359,E2 -17337.359} C_VEL
LIN {X 0,Y 313.969,Z 390.87,A -85,B 0,C 180,E1 -17337.76,E2 -17337.76} C_VEL
LIN {X 0,Y 306.719,Z 442.986,A -85,B 0,C 180,E1 -17340.012,E2 -17340.012} C_VEL
LIN {X 0,Y 303.943,Z 457.214,A -85,B 0,C 180,E1 -17340.854,E2 -17340.854} C_VEL
LIN {X 0,Y 300.57,Z 470.949,A -85,B 0,C 180,E1 -17341.928,E2 -17341.928} C_VEL
LIN {X 0,Y 297.403,Z 482.529,A -85,B 0,C 180,E1 -17343.13,E2 -17343.13} C_VEL
LIN {X 0,Y 293.696,Z 494.497,A -85,B 0,C 180,E1 -17344.674,E2 -17344.674} C_VEL
LIN {X 0,Y 290.743,Z 503.406,A -85,B 0,C 180,E1 -17346.114,E2 -17346.114} C_VEL
LIN {X 0,Y 287.212,Z 513.329,A -85,B 0,C 180,E1 -17348.088,E2 -17348.088} C_VEL
LIN {X 0,Y 283.88,Z 522.113,A -85,B 0,C 180,E1 -17350.266,E2 -17350.266} C_VEL
LIN {X 0,Y 281.658,Z 528.276,A -85,B 0,C 180,E1 -17352.2,E2 -17352.2} C_VEL
LIN {X 0,Y 279.297,Z 534.53,A -85,B 0,C 180,E1 -17354.678,E2 -17354.678} C_VEL
LIN {X 0,Y 277.635,Z 538.727,A -85,B 0,C 180,E1 -17356.83,E2 -17356.83} C_VEL
LIN {X 0,Y 276.871,Z 540.952,A -85,B 0,C 180,E1 -17358.282,E2 -17358.282} C_VEL
LIN {X 0,Y 276.227,Z 542.759,A -85,B 0,C 180,E1 -17359.739,E2 -17359.739} C_VEL
LIN {X 0,Y 275.775,Z 544.132,A -85,B 0,C 180,E1 -17361.203,E2 -17361.203} C_VEL
LIN {X 0,Y 275.333,Z 545.608,A -85,B 0,C 180,E1 -17364.138,E2 -17364.138} C_VEL
LIN {X 0,Y 275.329,Z 545.742,A -85,B 0,C 180,E1 -17365.607,E2 -17365.607} C_VEL
LIN {X 0,Y 275.408,Z 545.19,A -85,B 0,C 180,E1 -17368.536,E2 -17368.536} C_VEL
LIN {X 0,Y 275.576,Z 545.414,A -85,B 0,C 180,E1 -17369.999,E2 -17369.999} C_VEL
LIN {X 0,Y 275.467,Z 545.182,A -85,B 0,C 180,E1 -17371.46,E2 -17371.46} C_VEL
LIN {X 0,Y 275.422,Z 544.555,A -85,B 0,C 180,E1 -17372.924,E2 -17372.924} C_VEL
LIN {X 0,Y 275.346,Z 542.495,A -85,B 0,C 180,E1 -17375.47,E2 -17375.47} C_VEL
LIN {X 0,Y 275.553,Z 539.072,A -85,B 0,C 180,E1 -17378.062,E2 -17378.062} C_VEL
LIN {X 0,Y 275.972,Z 534.999,A -85,B 0,C 180,E1 -17380.267,E2 -17380.267} C_VEL
LIN {X 0,Y 276.882,Z 528.726,A -85,B 0,C 180,E1 -17382.831,E2 -17382.831} C_VEL
LIN {X 0,Y 278.187,Z 521.9,A -85,B 0,C 180,E1 -17385.006,E2 -17385.006} C_VEL
LIN {X 0,Y 279.612,Z 514.358,A -85,B 0,C 180,E1 -17386.942,E2 -17386.942} C_VEL
LIN {X 0,Y 281.252,Z 504.567,A -85,B 0,C 180,E1 -17388.955,E2 -17388.955} C_VEL
LIN {X 0,Y 282.969,Z 494.918,A -85,B 0,C 180,E1 -17390.536,E2 -17390.536} C_VEL
LIN {X 0,Y 284.747,Z 484.349,A -85,B 0,C 180,E1 -17391.918,E2 -17391.918} C_VEL
LIN {X 0,Y 286.363,Z 472.497,A -85,B 0,C 180,E1 -17393.119,E2 -17393.119} C_VEL
LIN {X 0,Y 287.848,Z 460.194,A -85,B 0,C 180,E1 -17394.042,E2 -17394.042} C_VEL
LIN {X 0,Y 288.924,Z 448.138,A -85,B 0,C 180,E1 -17394.678,E2 -17394.678} C_VEL
LIN {X 0,Y 289.599,Z 434.12,A -85,B 0,C 180,E1 -17395.124,E2 -17395.124} C_VEL
LIN {X 0,Y 290.844,Z 381.427,A -85,B 0,C 180,E1 -17396.416,E2 -17396.416} C_VEL
LIN {X 0,Y 286.77,Z 349.761,A -85,B 0,C 180,E1 -17397.686,E2 -17397.686} C_VEL
LIN {X 0,Y 284.457,Z 335.151,A -85,B 0,C 180,E1 -17398.336,E2 -17398.336} C_VEL
LIN {X 0,Y 279.865,Z 322.412,A -85,B 0,C 180,E1 -17399.203,E2 -17399.203} C_VEL
LIN {X 0,Y 278.906,Z 319.188,A -85,B 0,C 180,E1 -17399.447,E2 -17399.447} C_VEL
LIN {X 0,Y 277.332,Z 310.939,A -85,B 0,C 180,E1 -17402.15,E2 -17402.15} C_VEL
LIN {X 0,Y 277.303,Z 310.944,A -85,B 0,C 180,E1 -17405.805,E2 -17405.805} C_VEL
LIN {X 0,Y 277.232,Z 310.95,A -85,B 0,C 180,E1 -17409.326,E2 -17409.326} C_VEL
LIN {X 0,Y 277.204,Z 310.95,A -85,B 0,C 180,E1 -17413.197,E2 -17413.197} C_VEL
LIN {X 0,Y 277.187,Z 310.95,A -85,B 0,C 180,E1 -17417.329,E2 -17417.329} C_VEL
LIN {X 0,Y 277.215,Z 310.951,A -85,B 0,C 180,E1 -17421.803,E2 -17421.803} C_VEL
LIN {X 0,Y 277.27,Z 310.94,A -85,B 0,C 180,E1 -17424.339,E2 -17424.339} C_VEL
LIN {X 0,Y 277.23,Z 310.951,A -85,B 0,C 180,E1 -17427.834,E2 -17427.834} C_VEL
LIN {X 0,Y 277.211,Z 310.952,A -85,B 0,C 180,E1 -17431.204,E2 -17431.204} C_VEL
LIN {X 0,Y 277.23,Z 310.945,A -85,B 0,C 180,E1 -17434.471,E2 -17434.471} C_VEL
LIN {X 0,Y 277.247,Z 310.95,A -85,B 0,C 180,E1 -17437.652,E2 -17437.652} C_VEL
LIN {X 0,Y 277.277,Z 310.935,A -85,B 0,C 180,E1 -17440.761,E2 -17440.761} C_VEL
LIN {X 0,Y 277.401,Z 310.921,A -85,B 0,C 180,E1 -17445.324,E2 -17445.324} C_VEL
LIN {X 0,Y 277.449,Z 310.92,A -85,B 0,C 180,E1 -17449.787,E2 -17449.787} C_VEL
LIN {X 0,Y 277.59,Z 310.889,A -85,B 0,C 180,E1 -17452.727,E2 -17452.727} C_VEL
LIN {X 0,Y 277.796,Z 310.876,A -85,B 0,C 180,E1 -17458.55,E2 -17458.55} C_VEL
LIN {X 0,Y 277.801,Z 310.878,A -85,B 0,C 180,E1 -17461.45,E2 -17461.45} C_VEL
LIN {X 0,Y 277.591,Z 310.906,A -85,B 0,C 180,E1 -17467.273,E2 -17467.273} C_VEL
LIN {X 0,Y 277.449,Z 310.917,A -85,B 0,C 180,E1 -17470.214,E2 -17470.214} C_VEL
LIN {X 0,Y 277.401,Z 310.929,A -85,B 0,C 180,E1 -17474.676,E2 -17474.676} C_VEL
LIN {X 0,Y 277.309,Z 310.941,A -85,B 0,C 180,E1 -17479.237,E2 -17479.237} C_VEL
LIN {X 0,Y 277.28,Z 310.938,A -85,B 0,C 180,E1 -17483.925,E2 -17483.925} C_VEL
LIN {X 0,Y 277.274,Z 310.944,A -85,B 0,C 180,E1 -17487.488,E2 -17487.488} C_VEL
LIN {X 0,Y 277.241,Z 310.948,A -85,B 0,C 180,E1 -17490.474,E2 -17490.474} C_VEL
LIN {X 0,Y 277.24,Z 310.947,A -85,B 0,C 180,E1 -17493.897,E2 -17493.897} C_VEL
LIN {X 0,Y 277.261,Z 310.94,A -85,B 0,C 180,E1 -17497.471,E2 -17497.471} C_VEL
LIN {X 0,Y 277.204,Z 310.953,A -85,B 0,C 180,E1 -17501.238,E2 -17501.238} C_VEL
LIN {X 0,Y 277.196,Z 310.955,A -85,B 0,C 180,E1 -17505.228,E2 -17505.228} C_VEL
LIN {X 0,Y 277.219,Z 310.952,A -85,B 0,C 180,E1 -17509.514,E2 -17509.514} C_VEL
LIN {X 0,Y 277.268,Z 310.932,A -85,B 0,C 180,E1 -17512.533,E2 -17512.533} C_VEL
LIN {X 0,Y 277.244,Z 310.951,A -85,B 0,C 180,E1 -17516.106,E2 -17516.106} C_VEL
LIN {X 0,Y 277.338,Z 311.04,A -85,B 0,C 180,E1 -17520.615,E2 -17520.615} C_VEL
LIN {X 0,Y 278.382,Z 313.93,A -85,B 0,C 180,E1 -17520.821,E2 -17520.821} C_VEL
LIN {X 0,Y 286.412,Z 329.4,A -85,B 0,C 180,E1 -17522.155,E2 -17522.155} C_VEL
LIN {X 0,Y 292.46,Z 342.948,A -85,B 0,C 180,E1 -17523.154,E2 -17523.154} C_VEL
LIN {X 0,Y 290.391,Z 417.169,A -85,B 0,C 180,E1 -17524.992,E2 -17524.992} C_VEL
LIN {X 0,Y 289.665,Z 430.048,A -85,B 0,C 180,E1 -17525.547,E2 -17525.547} C_VEL
LIN {X 0,Y 288.543,Z 442.924,A -85,B 0,C 180,E1 -17526.401,E2 -17526.401} C_VEL
LIN {X 0,Y 287.122,Z 455.179,A -85,B 0,C 180,E1 -17527.516,E2 -17527.516} C_VEL
LIN {X 0,Y 285.428,Z 466.74,A -85,B 0,C 180,E1 -17528.895,E2 -17528.895} C_VEL
LIN {X 0,Y 283.932,Z 477.014,A -85,B 0,C 180,E1 -17530.475,E2 -17530.475} C_VEL
LIN {X 0,Y 282.188,Z 486.36,A -85,B 0,C 180,E1 -17532.238,E2 -17532.238} C_VEL
LIN {X 0,Y 280.583,Z 493.992,A -85,B 0,C 180,E1 -17534.008,E2 -17534.008} C_VEL
LIN {X 0,Y 279.151,Z 501.422,A -85,B 0,C 180,E1 -17536.164,E2 -17536.164} C_VEL
LIN {X 0,Y 277.913,Z 507.388,A -85,B 0,C 180,E1 -17538.33,E2 -17538.33} C_VEL
LIN {X 0,Y 276.955,Z 512.101,A -85,B 0,C 180,E1 -17540.508,E2 -17540.508} C_VEL
LIN {X 0,Y 276.336,Z 515.698,A -85,B 0,C 180,E1 -17542.696,E2 -17542.696} C_VEL
LIN {X 0,Y 276.005,Z 517.551,A -85,B 0,C 180,E1 -17544.156,E2 -17544.156} C_VEL
LIN {X 0,Y 275.771,Z 518.964,A -85,B 0,C 180,E1 -17545.617,E2 -17545.617} C_VEL
LIN {X 0,Y 275.437,Z 520.569,A -85,B 0,C 180,E1 -17548.539,E2 -17548.539} C_VEL
LIN {X 0,Y 275.417,Z 520.8,A -85,B 0,C 180,E1 -17550.001,E2 -17550.001} C_VEL
LIN {X 0,Y 275.556,Z 520.02,A -85,B 0,C 180,E1 -17552.925,E2 -17552.925} C_VEL
LIN {X 0,Y 275.768,Z 519.052,A -85,B 0,C 180,E1 -17554.386,E2 -17554.386} C_VEL
LIN {X 0,Y 276.001,Z 517.688,A -85,B 0,C 180,E1 -17555.847,E2 -17555.847} C_VEL
LIN {X 0,Y 276.483,Z 514.823,A -85,B 0,C 180,E1 -17558.038,E2 -17558.038} C_VEL
LIN {X 0,Y 277.175,Z 510.925,A -85,B 0,C 180,E1 -17560.225,E2 -17560.225} C_VEL
LIN {X 0,Y 278.258,Z 505.868,A -85,B 0,C 180,E1 -17562.399,E2 -17562.399} C_VEL
LIN {X 0,Y 279.577,Z 499.494,A -85,B 0,C 180,E1 -17564.561,E2 -17564.561} C_VEL
LIN {X 0,Y 281.158,Z 491.558,A -85,B 0,C 180,E1 -17566.707,E2 -17566.707} C_VEL
LIN {X 0,Y 282.831,Z 483.429,A -85,B 0,C 180,E1 -17568.472,E2 -17568.472} C_VEL
LIN {X 0,Y 284.477,Z 473.438,A -85,B 0,C 180,E1 -17570.236,E2 -17570.236} C_VEL
LIN {X 0,Y 286.201,Z 462.199,A -85,B 0,C 180,E1 -17571.804,E2 -17571.804} C_VEL
LIN {X 0,Y 287.751,Z 451.121,A -85,B 0,C 180,E1 -17573.005,E2 -17573.005} C_VEL
LIN {X 0,Y 288.93,Z 439.799,A -85,B 0,C 180,E1 -17573.95,E2 -17573.95} C_VEL
LIN {X 0,Y 289.935,Z 427.078,A -85,B 0,C 180,E1 -17574.718,E2 -17574.718} C_VEL
LIN {X 0,Y 290.62,Z 413.714,A -85,B 0,C 180,E1 -17575.229,E2 -17575.229} C_VEL
LIN {X 0,Y 292.535,Z 343.079,A -85,B 0,C 180,E1 -17576.958,E2 -17576.958} C_VEL
LIN {X 0,Y 284.686,Z 325.904,A -85,B 0,C 180,E1 -17578.254,E2 -17578.254} C_VEL
LIN {X 0,Y 277.554,Z 312.046,A -85,B 0,C 180,E1 -17579.458,E2 -17579.458} C_VEL
LIN {X 0,Y 277.328,Z 310.938,A -85,B 0,C 180,E1 -17579.575,E2 -17579.575} C_VEL
LIN {X 0,Y 277.259,Z 310.95,A -85,B 0,C 180,E1 -17583.896,E2 -17583.896} C_VEL
LIN {X 0,Y 277.286,Z 310.947,A -85,B 0,C 180,E1 -17587.468,E2 -17587.468} C_VEL
LIN {X 0,Y 277.232,Z 310.955,A -85,B 0,C 180,E1 -17591.234,E2 -17591.234} C_VEL
LIN {X 0,Y 277.225,Z 310.932,A -85,B 0,C 180,E1 -17595.223,E2 -17595.223} C_VEL
LIN {X 0,Y 277.228,Z 310.954,A -85,B 0,C 180,E1 -17599.513,E2 -17599.513} C_VEL
LIN {X 0,Y 277.27,Z 310.944,A -85,B 0,C 180,E1 -17602.531,E2 -17602.531} C_VEL
LIN {X 0,Y 277.252,Z 310.947,A -85,B 0,C 180,E1 -17606.105,E2 -17606.105} C_VEL
LIN {X 0,Y 277.267,Z 310.94,A -85,B 0,C 180,E1 -17609.539,E2 -17609.539} C_VEL
LIN {X 0,Y 277.362,Z 310.937,A -85,B 0,C 180,E1 -17612.864,E2 -17612.864} C_VEL
LIN {X 0,Y 277.39,Z 310.925,A -85,B 0,C 180,E1 -17615.8,E2 -17615.8} C_VEL
LIN {X 0,Y 284.355,Z 337.729,A -85,B 0,C 180,E1 -17617.191,E2 -17617.191} C_VEL
LIN {X 0,Y 284.423,Z 341.549,A -85,B 0,C 180,E1 -17617.347,E2 -17617.347} C_VEL
LIN {X 0,Y 283.171,Z 347.242,A -85,B 0,C 180,E1 -17617.529,E2 -17617.529} C_VEL
LIN {X 0,Y 277.371,Z 362.105,A -85,B 0,C 180,E1 -17617.933,E2 -17617.933} C_VEL
LIN {X 0,Y 276.367,Z 367.929,A -85,B 0,C 180,E1 -17618.142,E2 -17618.142} C_VEL
LIN {X 0,Y 274.421,Z 420.434,A -85,B 0,C 180,E1 -17620.31,E2 -17620.31} C_VEL
LIN {X 0,Y 273.714,Z 434.271,A -85,B 0,C 180,E1 -17621.182,E2 -17621.182} C_VEL
LIN {X 0,Y 272.949,Z 447.231,A -85,B 0,C 180,E1 -17622.309,E2 -17622.309} C_VEL
LIN {X 0,Y 272.179,Z 459.62,A -85,B 0,C 180,E1 -17623.692,E2 -17623.692} C_VEL
LIN {X 0,Y 271.216,Z 471.47,A -85,B 0,C 180,E1 -17625.365,E2 -17625.365} C_VEL
LIN {X 0,Y 270.273,Z 482.165,A -85,B 0,C 180,E1 -17627.23,E2 -17627.23} C_VEL
LIN {X 0,Y 269.604,Z 490.901,A -85,B 0,C 180,E1 -17629.106,E2 -17629.106} C_VEL
LIN {X 0,Y 269.028,Z 499.515,A -85,B 0,C 180,E1 -17631.361,E2 -17631.361} C_VEL
LIN {X 0,Y 268.685,Z 505.382,A -85,B 0,C 180,E1 -17633.241,E2 -17633.241} C_VEL
LIN {X 0,Y 268.46,Z 511.127,A -85,B 0,C 180,E1 -17635.495,E2 -17635.495} C_VEL
LIN {X 0,Y 268.345,Z 515.598,A -85,B 0,C 180,E1 -17637.748,E2 -17637.748} C_VEL
LIN {X 0,Y 268.297,Z 518.946,A -85,B 0,C 180,E1 -17640,E2 -17640} C_VEL
LIN {X 0,Y 268.41,Z 520.586,A -85,B 0,C 180,E1 -17641.5,E2 -17641.5} C_VEL
LIN {X 0,Y 268.626,Z 521.797,A -85,B 0,C 180,E1 -17642.999,E2 -17642.999} C_VEL
LIN {X 0,Y 268.911,Z 522.607,A -85,B 0,C 180,E1 -17644.497,E2 -17644.497} C_VEL
LIN {X 0,Y 269.22,Z 523,A -85,B 0,C 180,E1 -17645.994,E2 -17645.994} C_VEL
LIN {X 0,Y 269.711,Z 522.943,A -85,B 0,C 180,E1 -17647.486,E2 -17647.486} C_VEL
LIN {X 0,Y 270.502,Z 522.405,A -85,B 0,C 180,E1 -17649.138,E2 -17649.138} C_VEL
LIN {X 0,Y 272.209,Z 520.342,A -85,B 0,C 180,E1 -17651.92,E2 -17651.92} C_VEL
LIN {X 0,Y 273.979,Z 517.604,A -85,B 0,C 180,E1 -17654.104,E2 -17654.104} C_VEL
LIN {X 0,Y 276.067,Z 513.847,A -85,B 0,C 180,E1 -17656.262,E2 -17656.262} C_VEL
LIN {X 0,Y 278.537,Z 508.997,A -85,B 0,C 180,E1 -17658.385,E2 -17658.385} C_VEL
LIN {X 0,Y 281.373,Z 502.927,A -85,B 0,C 180,E1 -17660.468,E2 -17660.468} C_VEL
LIN {X 0,Y 284.679,Z 495.411,A -85,B 0,C 180,E1 -17662.498,E2 -17662.498} C_VEL
LIN {X 0,Y 288.347,Z 486.241,A -85,B 0,C 180,E1 -17664.478,E2 -17664.478} C_VEL
LIN {X 0,Y 292.405,Z 474.829,A -85,B 0,C 180,E1 -17666.401,E2 -17666.401} C_VEL
LIN {X 0,Y 295.498,Z 464.935,A -85,B 0,C 180,E1 -17667.745,E2 -17667.745} C_VEL
LIN {X 0,Y 299.131,Z 451.522,A -85,B 0,C 180,E1 -17669.177,E2 -17669.177} C_VEL
LIN {X 0,Y 301.954,Z 438.854,A -85,B 0,C 180,E1 -17670.22,E2 -17670.22} C_VEL
LIN {X 0,Y 304.455,Z 425.202,A -85,B 0,C 180,E1 -17671.05,E2 -17671.05} C_VEL
LIN {X 0,Y 312.159,Z 374.535,A -85,B 0,C 180,E1 -17673.292,E2 -17673.292} C_VEL
LIN {X 0,Y 309.496,Z 369.157,A -85,B 0,C 180,E1 -17674.935,E2 -17674.935} C_VEL
LIN {X 0,Y 307.539,Z 365.701,A -85,B 0,C 180,E1 -17676.309,E2 -17676.309} C_VEL
LIN {X 0,Y 306.225,Z 363.515,A -85,B 0,C 180,E1 -17677.378,E2 -17677.378} C_VEL
LIN {X 0,Y 304.259,Z 360.517,A -85,B 0,C 180,E1 -17679.35,E2 -17679.35} C_VEL
LIN {X 0,Y 302.339,Z 358.483,A -85,B 0,C 180,E1 -17682.386,E2 -17682.386} C_VEL
LIN {X 0,Y 302.002,Z 358.081,A -85,B 0,C 180,E1 -17683.827,E2 -17683.827} C_VEL
LIN {X 0,Y 302.048,Z 358.983,A -85,B 0,C 180,E1 -17686.162,E2 -17686.162} C_VEL
LIN {X 0,Y 302.763,Z 361.679,A -85,B 0,C 180,E1 -17688.44,E2 -17688.44} C_VEL
LIN {X 0,Y 304.885,Z 366.378,A -85,B 0,C 180,E1 -17691.213,E2 -17691.213} C_VEL
LIN {X 0,Y 307.165,Z 372.302,A -85,B 0,C 180,E1 -17693.346,E2 -17693.346} C_VEL
LIN {X 0,Y 309.045,Z 377.545,A -85,B 0,C 180,E1 -17694.797,E2 -17694.797} C_VEL
LIN {X 0,Y 310.05,Z 380.849,A -85,B 0,C 180,E1 -17695.536,E2 -17695.536} C_VEL
LIN {X 0,Y 310.232,Z 390.523,A -85,B 0,C 180,E1 -17696.556,E2 -17696.556} C_VEL
LIN {X 0,Y 309.933,Z 393.824,A -85,B 0,C 180,E1 -17696.77,E2 -17696.77} C_VEL
LIN {X 0,Y 302.657,Z 442.26,A -85,B 0,C 180,E1 -17698.89,E2 -17698.89} C_VEL
LIN {X 0,Y 299.719,Z 456.337,A -85,B 0,C 180,E1 -17699.724,E2 -17699.724} C_VEL
LIN {X 0,Y 295.937,Z 470.804,A -85,B 0,C 180,E1 -17700.866,E2 -17700.866} C_VEL
LIN {X 0,Y 292.166,Z 483.549,A -85,B 0,C 180,E1 -17702.22,E2 -17702.22} C_VEL
LIN {X 0,Y 288.278,Z 495.104,A -85,B 0,C 180,E1 -17703.775,E2 -17703.775} C_VEL
LIN {X 0,Y 284.484,Z 505.564,A -85,B 0,C 180,E1 -17705.555,E2 -17705.555} C_VEL
LIN {X 0,Y 280.809,Z 514.989,A -85,B 0,C 180,E1 -17707.561,E2 -17707.561} C_VEL
LIN {X 0,Y 277.35,Z 523.203,A -85,B 0,C 180,E1 -17709.753,E2 -17709.753} C_VEL
LIN {X 0,Y 274.614,Z 530.097,A -85,B 0,C 180,E1 -17712.114,E2 -17712.114} C_VEL
LIN {X 0,Y 272.468,Z 535.112,A -85,B 0,C 180,E1 -17714.285,E2 -17714.285} C_VEL
LIN {X 0,Y 270.714,Z 539.055,A -85,B 0,C 180,E1 -17716.487,E2 -17716.487} C_VEL
LIN {X 0,Y 269.905,Z 541.143,A -85,B 0,C 180,E1 -17717.975,E2 -17717.975} C_VEL
LIN {X 0,Y 268.734,Z 544.005,A -85,B 0,C 180,E1 -17720.971,E2 -17720.971} C_VEL
LIN {X 0,Y 268.244,Z 545.274,A -85,B 0,C 180,E1 -17723.983,E2 -17723.983} C_VEL
LIN {X 0,Y 268.251,Z 545.262,A -85,B 0,C 180,E1 -17725.491,E2 -17725.491} C_VEL
LIN {X 0,Y 268.287,Z 544.825,A -85,B 0,C 180,E1 -17726.995,E2 -17726.995} C_VEL
LIN {X 0,Y 268.484,Z 545.098,A -85,B 0,C 180,E1 -17729.998,E2 -17729.998} C_VEL
LIN {X 0,Y 268.383,Z 544.866,A -85,B 0,C 180,E1 -17731.499,E2 -17731.499} C_VEL
LIN {X 0,Y 268.322,Z 544.237,A -85,B 0,C 180,E1 -17733.001,E2 -17733.001} C_VEL
LIN {X 0,Y 268.244,Z 542.411,A -85,B 0,C 180,E1 -17735.375,E2 -17735.375} C_VEL
LIN {X 0,Y 268.499,Z 538.754,A -85,B 0,C 180,E1 -17738.276,E2 -17738.276} C_VEL
LIN {X 0,Y 268.938,Z 534.68,A -85,B 0,C 180,E1 -17740.539,E2 -17740.539} C_VEL
LIN {X 0,Y 269.947,Z 528.409,A -85,B 0,C 180,E1 -17743.166,E2 -17743.166} C_VEL
LIN {X 0,Y 271.264,Z 521.581,A -85,B 0,C 180,E1 -17745.399,E2 -17745.399} C_VEL
LIN {X 0,Y 272.861,Z 513.721,A -85,B 0,C 180,E1 -17747.453,E2 -17747.453} C_VEL
LIN {X 0,Y 274.518,Z 504.253,A -85,B 0,C 180,E1 -17749.438,E2 -17749.438} C_VEL
LIN {X 0,Y 276.328,Z 494.608,A -85,B 0,C 180,E1 -17751.052,E2 -17751.052} C_VEL
LIN {X 0,Y 278.167,Z 484.041,A -85,B 0,C 180,E1 -17752.465,E2 -17752.465} C_VEL
LIN {X 0,Y 279.838,Z 472.196,A -85,B 0,C 180,E1 -17753.691,E2 -17753.691} C_VEL
LIN {X 0,Y 281.373,Z 459.901,A -85,B 0,C 180,E1 -17754.632,E2 -17754.632} C_VEL
LIN {X 0,Y 282.576,Z 447.092,A -85,B 0,C 180,E1 -17755.307,E2 -17755.307} C_VEL
LIN {X 0,Y 283.264,Z 431.479,A -85,B 0,C 180,E1 -17755.793,E2 -17755.793} C_VEL
LIN {X 0,Y 284.505,Z 382.326,A -85,B 0,C 180,E1 -17757.021,E2 -17757.021} C_VEL
LIN {X 0,Y 280.486,Z 350.915,A -85,B 0,C 180,E1 -17758.323,E2 -17758.323} C_VEL
LIN {X 0,Y 278.411,Z 337.35,A -85,B 0,C 180,E1 -17758.94,E2 -17758.94} C_VEL
LIN {X 0,Y 272.573,Z 321.404,A -85,B 0,C 180,E1 -17760.086,E2 -17760.086} C_VEL
LIN {X 0,Y 271.295,Z 317.225,A -85,B 0,C 180,E1 -17760.452,E2 -17760.452} C_VEL
LIN {X 0,Y 270.273,Z 311.818,A -85,B 0,C 180,E1 -17762.266,E2 -17762.266} C_VEL
LIN {X 0,Y 270.224,Z 311.821,A -85,B 0,C 180,E1 -17766.738,E2 -17766.738} C_VEL
LIN {X 0,Y 270.164,Z 311.828,A -85,B 0,C 180,E1 -17771.027,E2 -17771.027} C_VEL
LIN {X 0,Y 270.145,Z 311.831,A -85,B 0,C 180,E1 -17774.619,E2 -17774.619} C_VEL
LIN {X 0,Y 270.145,Z 311.827,A -85,B 0,C 180,E1 -17777.436,E2 -17777.436} C_VEL
LIN {X 0,Y 270.145,Z 311.827,A -85,B 0,C 180,E1 -17781.363,E2 -17781.363} C_VEL
LIN {X 0,Y 270.191,Z 311.822,A -85,B 0,C 180,E1 -17785.093,E2 -17785.093} C_VEL
LIN {X 0,Y 270.164,Z 311.829,A -85,B 0,C 180,E1 -17789.14,E2 -17789.14} C_VEL
LIN {X 0,Y 270.181,Z 311.829,A -85,B 0,C 180,E1 -17792.176,E2 -17792.176} C_VEL
LIN {X 0,Y 270.181,Z 311.827,A -85,B 0,C 180,E1 -17795.56,E2 -17795.56} C_VEL
LIN {X 0,Y 270.216,Z 311.814,A -85,B 0,C 180,E1 -17800.238,E2 -17800.238} C_VEL
LIN {X 0,Y 270.36,Z 311.794,A -85,B 0,C 180,E1 -17804.933,E2 -17804.933} C_VEL
LIN {X 0,Y 270.401,Z 311.799,A -85,B 0,C 180,E1 -17809.517,E2 -17809.517} C_VEL
LIN {X 0,Y 270.552,Z 311.766,A -85,B 0,C 180,E1 -17812.537,E2 -17812.537} C_VEL
LIN {X 0,Y 270.761,Z 311.751,A -85,B 0,C 180,E1 -17818.513,E2 -17818.513} C_VEL
LIN {X 0,Y 270.766,Z 311.754,A -85,B 0,C 180,E1 -17821.487,E2 -17821.487} C_VEL
LIN {X 0,Y 270.553,Z 311.781,A -85,B 0,C 180,E1 -17827.463,E2 -17827.463} C_VEL
LIN {X 0,Y 270.402,Z 311.795,A -85,B 0,C 180,E1 -17830.483,E2 -17830.483} C_VEL
LIN {X 0,Y 270.36,Z 311.802,A -85,B 0,C 180,E1 -17835.067,E2 -17835.067} C_VEL
LIN {X 0,Y 270.25,Z 311.818,A -85,B 0,C 180,E1 -17839.76,E2 -17839.76} C_VEL
LIN {X 0,Y 270.22,Z 311.815,A -85,B 0,C 180,E1 -17844.591,E2 -17844.591} C_VEL
LIN {X 0,Y 270.202,Z 311.825,A -85,B 0,C 180,E1 -17847.917,E2 -17847.917} C_VEL
LIN {X 0,Y 270.167,Z 311.822,A -85,B 0,C 180,E1 -17851.351,E2 -17851.351} C_VEL
LIN {X 0,Y 270.196,Z 311.828,A -85,B 0,C 180,E1 -17854.907,E2 -17854.907} C_VEL
LIN {X 0,Y 270.192,Z 311.823,A -85,B 0,C 180,E1 -17858.712,E2 -17858.712} C_VEL
LIN {X 0,Y 270.166,Z 311.827,A -85,B 0,C 180,E1 -17862.56,E2 -17862.56} C_VEL
LIN {X 0,Y 270.161,Z 311.828,A -85,B 0,C 180,E1 -17866.752,E2 -17866.752} C_VEL
LIN {X 0,Y 270.17,Z 311.83,A -85,B 0,C 180,E1 -17869.436,E2 -17869.436} C_VEL
LIN {X 0,Y 270.224,Z 311.812,A -85,B 0,C 180,E1 -17873.732,E2 -17873.732} C_VEL
LIN {X 0,Y 270.2,Z 311.823,A -85,B 0,C 180,E1 -17876.894,E2 -17876.894} C_VEL
LIN {X 0,Y 270.242,Z 311.82,A -85,B 0,C 180,E1 -17879.765,E2 -17879.765} C_VEL
LIN {X 0,Y 271.285,Z 314.707,A -85,B 0,C 180,E1 -17879.996,E2 -17879.996} C_VEL
LIN {X 0,Y 279.758,Z 330.774,A -85,B 0,C 180,E1 -17881.466,E2 -17881.466} C_VEL
LIN {X 0,Y 286.096,Z 344.758,A -85,B 0,C 180,E1 -17882.551,E2 -17882.551} C_VEL
LIN {X 0,Y 285.126,Z 379.997,A -85,B 0,C 180,E1 -17883.431,E2 -17883.431} C_VEL
LIN {X 0,Y 283.955,Z 418.745,A -85,B 0,C 180,E1 -17884.434,E2 -17884.434} C_VEL
LIN {X 0,Y 283.09,Z 431.842,A -85,B 0,C 180,E1 -17885.038,E2 -17885.038} C_VEL
LIN {X 0,Y 281.865,Z 445.368,A -85,B 0,C 180,E1 -17886.002,E2 -17886.002} C_VEL
LIN {X 0,Y 280.393,Z 457.112,A -85,B 0,C 180,E1 -17887.14,E2 -17887.14} C_VEL
LIN {X 0,Y 278.63,Z 468.298,A -85,B 0,C 180,E1 -17888.549,E2 -17888.549} C_VEL
LIN {X 0,Y 277.015,Z 478.809,A -85,B 0,C 180,E1 -17890.243,E2 -17890.243} C_VEL
LIN {X 0,Y 275.129,Z 488.299,A -85,B 0,C 180,E1 -17892.151,E2 -17892.151} C_VEL
LIN {X 0,Y 273.525,Z 495.637,A -85,B 0,C 180,E1 -17893.967,E2 -17893.967} C_VEL
LIN {X 0,Y 272.047,Z 502.826,A -85,B 0,C 180,E1 -17896.176,E2 -17896.176} C_VEL
LIN {X 0,Y 270.586,Z 509.423,A -85,B 0,C 180,E1 -17898.769,E2 -17898.769} C_VEL
LIN {X 0,Y 269.723,Z 513.745,A -85,B 0,C 180,E1 -17901.007,E2 -17901.007} C_VEL
LIN {X 0,Y 269.229,Z 516.331,A -85,B 0,C 180,E1 -17902.731,E2 -17902.731} C_VEL
LIN {X 0,Y 268.719,Z 519.281,A -85,B 0,C 180,E1 -17905.501,E2 -17905.501} C_VEL
LIN {X 0,Y 268.36,Z 520.885,A -85,B 0,C 180,E1 -17908.501,E2 -17908.501} C_VEL
LIN {X 0,Y 268.336,Z 521.117,A -85,B 0,C 180,E1 -17910.002,E2 -17910.002} C_VEL
LIN {X 0,Y 268.49,Z 520.335,A -85,B 0,C 180,E1 -17913.002,E2 -17913.002} C_VEL
LIN {X 0,Y 268.716,Z 519.368,A -85,B 0,C 180,E1 -17914.502,E2 -17914.502} C_VEL
LIN {X 0,Y 269.197,Z 516.574,A -85,B 0,C 180,E1 -17917.216,E2 -17917.216} C_VEL
LIN {X 0,Y 269.909,Z 512.637,A -85,B 0,C 180,E1 -17919.746,E2 -17919.746} C_VEL
LIN {X 0,Y 270.894,Z 507.984,A -85,B 0,C 180,E1 -17921.98,E2 -17921.98} C_VEL
LIN {X 0,Y 272.191,Z 502.085,A -85,B 0,C 180,E1 -17924.2,E2 -17924.2} C_VEL
LIN {X 0,Y 273.725,Z 494.736,A -85,B 0,C 180,E1 -17926.407,E2 -17926.407} C_VEL
LIN {X 0,Y 275.466,Z 487.192,A -85,B 0,C 180,E1 -17928.214,E2 -17928.214} C_VEL
LIN {X 0,Y 277.185,Z 477.79,A -85,B 0,C 180,E1 -17930.056,E2 -17930.056} C_VEL
LIN {X 0,Y 278.805,Z 467.816,A -85,B 0,C 180,E1 -17931.634,E2 -17931.634} C_VEL
LIN {X 0,Y 280.508,Z 456.514,A -85,B 0,C 180,E1 -17933.048,E2 -17933.048} C_VEL
LIN {X 0,Y 281.951,Z 444.541,A -85,B 0,C 180,E1 -17934.189,E2 -17934.189} C_VEL
LIN {X 0,Y 283.188,Z 431.451,A -85,B 0,C 180,E1 -17935.103,E2 -17935.103} C_VEL
LIN {X 0,Y 283.979,Z 419.342,A -85,B 0,C 180,E1 -17935.666,E2 -17935.666} C_VEL
LIN {X 0,Y 285.182,Z 380.153,A -85,B 0,C 180,E1 -17936.684,E2 -17936.684} C_VEL
LIN {X 0,Y 286.172,Z 344.883,A -85,B 0,C 180,E1 -17937.562,E2 -17937.562} C_VEL
LIN {X 0,Y 278.707,Z 328.728,A -85,B 0,C 180,E1 -17938.839,E2 -17938.839} C_VEL
LIN {X 0,Y 271.528,Z 315.086,A -85,B 0,C 180,E1 -17940.093,E2 -17940.093} C_VEL
LIN {X 0,Y 270.298,Z 312.164,A -85,B 0,C 180,E1 -17940.334,E2 -17940.334} C_VEL
LIN {X 0,Y 270.232,Z 311.824,A -85,B 0,C 180,E1 -17940.394,E2 -17940.394} C_VEL
LIN {X 0,Y 270.22,Z 311.825,A -85,B 0,C 180,E1 -17944.904,E2 -17944.904} C_VEL
LIN {X 0,Y 270.227,Z 311.827,A -85,B 0,C 180,E1 -17948.718,E2 -17948.718} C_VEL
LIN {X 0,Y 270.197,Z 311.83,A -85,B 0,C 180,E1 -17952.555,E2 -17952.555} C_VEL
LIN {X 0,Y 270.177,Z 311.808,A -85,B 0,C 180,E1 -17956.75,E2 -17956.75} C_VEL
LIN {X 0,Y 270.203,Z 311.828,A -85,B 0,C 180,E1 -17961.29,E2 -17961.29} C_VEL
LIN {X 0,Y 270.207,Z 311.826,A -85,B 0,C 180,E1 -17965.095,E2 -17965.095} C_VEL
LIN {X 0,Y 270.206,Z 311.818,A -85,B 0,C 180,E1 -17969.131,E2 -17969.131} C_VEL
LIN {X 0,Y 270.27,Z 311.817,A -85,B 0,C 180,E1 -17972.146,E2 -17972.146} C_VEL
LIN {X 0,Y 270.334,Z 311.803,A -85,B 0,C 180,E1 -17975.538,E2 -17975.538} C_VEL
LIN {X 0,Y 277.437,Z 338.899,A -85,B 0,C 180,E1 -17976.978,E2 -17976.978} C_VEL
LIN {X 0,Y 276.367,Z 367.929,A -85,B 0,C 180,E1 -17978.142,E2 -17978.142} C_VEL
LIN {X 0,Y 275.502,Z 373.679,A -85,B 0,C 180,E1 -17978.355,E2 -17978.355} C_VEL
LIN {X 0,Y 269.062,Z 392.224,A -85,B 0,C 180,E1 -17978.956,E2 -17978.956} C_VEL
LIN {X 0,Y 268.21,Z 397.973,A -85,B 0,C 180,E1 -17979.181,E2 -17979.181} C_VEL
LIN {X 0,Y 267.27,Z 422.058,A -85,B 0,C 180,E1 -17980.261,E2 -17980.261} C_VEL
LIN {X 0,Y 266.645,Z 434.265,A -85,B 0,C 180,E1 -17981.063,E2 -17981.063} C_VEL
LIN {X 0,Y 265.852,Z 447.494,A -85,B 0,C 180,E1 -17982.244,E2 -17982.244} C_VEL
LIN {X 0,Y 265.089,Z 459.675,A -85,B 0,C 180,E1 -17983.639,E2 -17983.639} C_VEL
LIN {X 0,Y 264.106,Z 471.543,A -85,B 0,C 180,E1 -17985.357,E2 -17985.357} C_VEL
LIN {X 0,Y 263.159,Z 482.276,A -85,B 0,C 180,E1 -17987.272,E2 -17987.272} C_VEL
LIN {X 0,Y 262.396,Z 492.644,A -85,B 0,C 180,E1 -17989.584,E2 -17989.584} C_VEL
LIN {X 0,Y 261.833,Z 500.975,A -85,B 0,C 180,E1 -17991.899,E2 -17991.899} C_VEL
LIN {X 0,Y 261.462,Z 507.829,A -85,B 0,C 180,E1 -17994.283,E2 -17994.283} C_VEL
LIN {X 0,Y 261.362,Z 513.775,A -85,B 0,C 180,E1 -17996.917,E2 -17996.917} C_VEL
LIN {X 0,Y 261.201,Z 517.691,A -85,B 0,C 180,E1 -17999.229,E2 -17999.229} C_VEL
LIN {X 0,Y 261.334,Z 520.553,A -85,B 0,C 180,E1 -18001.541,E2 -18001.541} C_VEL
LIN {X 0,Y 261.558,Z 521.906,A -85,B 0,C 180,E1 -18003.08,E2 -18003.08} C_VEL
LIN {X 0,Y 261.857,Z 522.82,A -85,B 0,C 180,E1 -18004.618,E2 -18004.618} C_VEL
LIN {X 0,Y 262.174,Z 523.341,A -85,B 0,C 180,E1 -18006.155,E2 -18006.155} C_VEL
LIN {X 0,Y 262.701,Z 523.461,A -85,B 0,C 180,E1 -18007.687,E2 -18007.687} C_VEL
LIN {X 0,Y 263.438,Z 523.143,A -85,B 0,C 180,E1 -18009.211,E2 -18009.211} C_VEL
LIN {X 0,Y 264.379,Z 522.396,A -85,B 0,C 180,E1 -18010.724,E2 -18010.724} C_VEL
LIN {X 0,Y 266.417,Z 519.749,A -85,B 0,C 180,E1 -18013.734,E2 -18013.734} C_VEL
LIN {X 0,Y 268.645,Z 516.57,A -85,B 0,C 180,E1 -18015.944,E2 -18015.944} C_VEL
LIN {X 0,Y 271.091,Z 512.396,A -85,B 0,C 180,E1 -18018.125,E2 -18018.125} C_VEL
LIN {X 0,Y 274.493,Z 506.065,A -85,B 0,C 180,E1 -18020.613,E2 -18020.613} C_VEL
LIN {X 0,Y 278.451,Z 497.972,A -85,B 0,C 180,E1 -18023.03,E2 -18023.03} C_VEL
LIN {X 0,Y 282.309,Z 489.276,A -85,B 0,C 180,E1 -18025.037,E2 -18025.037} C_VEL
LIN {X 0,Y 286.559,Z 478.623,A -85,B 0,C 180,E1 -18026.983,E2 -18026.983} C_VEL
LIN {X 0,Y 290.323,Z 467.715,A -85,B 0,C 180,E1 -18028.561,E2 -18028.561} C_VEL
LIN {X 0,Y 293.978,Z 455.723,A -85,B 0,C 180,E1 -18029.937,E2 -18029.937} C_VEL
LIN {X 0,Y 296.899,Z 444.268,A -85,B 0,C 180,E1 -18030.976,E2 -18030.976} C_VEL
LIN {X 0,Y 299.558,Z 431.987,A -85,B 0,C 180,E1 -18031.831,E2 -18031.831} C_VEL
LIN {X 0,Y 302.049,Z 417.235,A -85,B 0,C 180,E1 -18032.585,E2 -18032.585} C_VEL
LIN {X 0,Y 308.361,Z 378.551,A -85,B 0,C 180,E1 -18034.31,E2 -18034.31} C_VEL
LIN {X 0,Y 305.85,Z 373.309,A -85,B 0,C 180,E1 -18036.105,E2 -18036.105} C_VEL
LIN {X 0,Y 304.048,Z 370.12,A -85,B 0,C 180,E1 -18037.624,E2 -18037.624} C_VEL
LIN {X 0,Y 302.284,Z 367.289,A -85,B 0,C 180,E1 -18039.506,E2 -18039.506} C_VEL
LIN {X 0,Y 300.418,Z 365.196,A -85,B 0,C 180,E1 -18042.721,E2 -18042.721} C_VEL
LIN {X 0,Y 300.259,Z 364.961,A -85,B 0,C 180,E1 -18043.48,E2 -18043.48} C_VEL
LIN {X 0,Y 300.141,Z 365.567,A -85,B 0,C 180,E1 -18045.652,E2 -18045.652} C_VEL
LIN {X 0,Y 300.389,Z 366.819,A -85,B 0,C 180,E1 -18047.02,E2 -18047.02} C_VEL
LIN {X 0,Y 301.855,Z 371.094,A -85,B 0,C 180,E1 -18049.928,E2 -18049.928} C_VEL
LIN {X 0,Y 302.674,Z 373.091,A -85,B 0,C 180,E1 -18050.932,E2 -18050.932} C_VEL
LIN {X 0,Y 304.455,Z 378.133,A -85,B 0,C 180,E1 -18052.788,E2 -18052.788} C_VEL
LIN {X 0,Y 306.018,Z 383.014,A -85,B 0,C 180,E1 -18054.17,E2 -18054.17} C_VEL
LIN {X 0,Y 306.661,Z 385.396,A -85,B 0,C 180,E1 -18054.713,E2 -18054.713} C_VEL
LIN {X 0,Y 306.539,Z 393.829,A -85,B 0,C 180,E1 -18055.585,E2 -18055.585} C_VEL
LIN {X 0,Y 298.635,Z 442.763,A -85,B 0,C 180,E1 -18057.778,E2 -18057.778} C_VEL
LIN {X 0,Y 295.427,Z 456.863,A -85,B 0,C 180,E1 -18058.64,E2 -18058.64} C_VEL
LIN {X 0,Y 291.985,Z 469.398,A -85,B 0,C 180,E1 -18059.637,E2 -18059.637} C_VEL
LIN {X 0,Y 287.86,Z 482.233,A -85,B 0,C 180,E1 -18060.97,E2 -18060.97} C_VEL
LIN {X 0,Y 283.742,Z 493.84,A -85,B 0,C 180,E1 -18062.526,E2 -18062.526} C_VEL
LIN {X 0,Y 279.602,Z 504.359,A -85,B 0,C 180,E1 -18064.303,E2 -18064.303} C_VEL
LIN {X 0,Y 275.64,Z 513.876,A -85,B 0,C 180,E1 -18066.322,E2 -18066.322} C_VEL
LIN {X 0,Y 271.552,Z 522.871,A -85,B 0,C 180,E1 -18068.755,E2 -18068.755} C_VEL
LIN {X 0,Y 268.715,Z 529.119,A -85,B 0,C 180,E1 -18070.916,E2 -18070.916} C_VEL
LIN {X 0,Y 266.379,Z 534.196,A -85,B 0,C 180,E1 -18073.128,E2 -18073.128} C_VEL
LIN {X 0,Y 264.384,Z 538.224,A -85,B 0,C 180,E1 -18075.371,E2 -18075.371} C_VEL
LIN {X 0,Y 262.934,Z 541.264,A -85,B 0,C 180,E1 -18077.651,E2 -18077.651} C_VEL
LIN {X 0,Y 261.711,Z 543.893,A -85,B 0,C 180,E1 -18080.726,E2 -18080.726} C_VEL
LIN {X 0,Y 261.332,Z 544.578,A -85,B 0,C 180,E1 -18082.271,E2 -18082.271} C_VEL
LIN {X 0,Y 261.175,Z 544.728,A -85,B 0,C 180,E1 -18085.368,E2 -18085.368} C_VEL
LIN {X 0,Y 261.218,Z 544.192,A -85,B 0,C 180,E1 -18086.914,E2 -18086.914} C_VEL
LIN {X 0,Y 261.394,Z 544.781,A -85,B 0,C 180,E1 -18089.998,E2 -18089.998} C_VEL
LIN {X 0,Y 261.3,Z 544.549,A -85,B 0,C 180,E1 -18091.54,E2 -18091.54} C_VEL
LIN {X 0,Y 261.225,Z 543.919,A -85,B 0,C 180,E1 -18093.083,E2 -18093.083} C_VEL
LIN {X 0,Y 261.144,Z 542.324,A -85,B 0,C 180,E1 -18095.277,E2 -18095.277} C_VEL
LIN {X 0,Y 261.439,Z 538.435,A -85,B 0,C 180,E1 -18098.501,E2 -18098.501} C_VEL
LIN {X 0,Y 261.923,Z 534.361,A -85,B 0,C 180,E1 -18100.824,E2 -18100.824} C_VEL
LIN {X 0,Y 263.015,Z 528.091,A -85,B 0,C 180,E1 -18103.52,E2 -18103.52} C_VEL
LIN {X 0,Y 264.375,Z 521.263,A -85,B 0,C 180,E1 -18105.81,E2 -18105.81} C_VEL
LIN {X 0,Y 265.922,Z 514.103,A -85,B 0,C 180,E1 -18107.744,E2 -18107.744} C_VEL
LIN {X 0,Y 267.434,Z 505.875,A -85,B 0,C 180,E1 -18109.575,E2 -18109.575} C_VEL
LIN {X 0,Y 269.474,Z 495.461,A -85,B 0,C 180,E1 -18111.414,E2 -18111.414} C_VEL
LIN {X 0,Y 271.601,Z 483.733,A -85,B 0,C 180,E1 -18113.038,E2 -18113.038} C_VEL
LIN {X 0,Y 273.343,Z 471.893,A -85,B 0,C 180,E1 -18114.29,E2 -18114.29} C_VEL
LIN {X 0,Y 274.912,Z 459.606,A -85,B 0,C 180,E1 -18115.251,E2 -18115.251} C_VEL
LIN {X 0,Y 276.152,Z 446.989,A -85,B 0,C 180,E1 -18115.931,E2 -18115.931} C_VEL
LIN {X 0,Y 276.875,Z 432.04,A -85,B 0,C 180,E1 -18116.411,E2 -18116.411} C_VEL
LIN {X 0,Y 278.152,Z 382.849,A -85,B 0,C 180,E1 -18117.669,E2 -18117.669} C_VEL
LIN {X 0,Y 273.805,Z 348.874,A -85,B 0,C 180,E1 -18119.132,E2 -18119.132} C_VEL
LIN {X 0,Y 272.363,Z 339.53,A -85,B 0,C 180,E1 -18119.575,E2 -18119.575} C_VEL
LIN {X 0,Y 265.078,Z 319.665,A -85,B 0,C 180,E1 -18121.093,E2 -18121.093} C_VEL
LIN {X 0,Y 263.694,Z 315.318,A -85,B 0,C 180,E1 -18121.475,E2 -18121.475} C_VEL
LIN {X 0,Y 263.249,Z 312.693,A -85,B 0,C 180,E1 -18122.383,E2 -18122.383} C_VEL
LIN {X 0,Y 263.189,Z 312.697,A -85,B 0,C 180,E1 -18126.765,E2 -18126.765} C_VEL
LIN {X 0,Y 263.119,Z 312.708,A -85,B 0,C 180,E1 -18131.592,E2 -18131.592} C_VEL
LIN {X 0,Y 263.092,Z 312.707,A -85,B 0,C 180,E1 -18136.009,E2 -18136.009} C_VEL
LIN {X 0,Y 263.066,Z 312.708,A -85,B 0,C 180,E1 -18140.12,E2 -18140.12} C_VEL
LIN {X 0,Y 263.147,Z 312.701,A -85,B 0,C 180,E1 -18144.015,E2 -18144.015} C_VEL
LIN {X 0,Y 263.119,Z 312.71,A -85,B 0,C 180,E1 -18147.71,E2 -18147.71} C_VEL
LIN {X 0,Y 263.129,Z 312.71,A -85,B 0,C 180,E1 -18151.809,E2 -18151.809} C_VEL
LIN {X 0,Y 263.116,Z 312.708,A -85,B 0,C 180,E1 -18156.381,E2 -18156.381} C_VEL
LIN {X 0,Y 263.201,Z 312.69,A -85,B 0,C 180,E1 -18159.688,E2 -18159.688} C_VEL
LIN {X 0,Y 263.302,Z 312.671,A -85,B 0,C 180,E1 -18164.519,E2 -18164.519} C_VEL
LIN {X 0,Y 263.344,Z 312.681,A -85,B 0,C 180,E1 -18169.233,E2 -18169.233} C_VEL
LIN {X 0,Y 263.516,Z 312.643,A -85,B 0,C 180,E1 -18172.337,E2 -18172.337} C_VEL
LIN {X 0,Y 263.725,Z 312.628,A -85,B 0,C 180,E1 -18178.473,E2 -18178.473} C_VEL
LIN {X 0,Y 263.728,Z 312.63,A -85,B 0,C 180,E1 -18181.527,E2 -18181.527} C_VEL
LIN {X 0,Y 263.517,Z 312.657,A -85,B 0,C 180,E1 -18187.663,E2 -18187.663} C_VEL
LIN {X 0,Y 263.341,Z 312.676,A -85,B 0,C 180,E1 -18190.767,E2 -18190.767} C_VEL
LIN {X 0,Y 263.302,Z 312.678,A -85,B 0,C 180,E1 -18195.481,E2 -18195.481} C_VEL
LIN {X 0,Y 263.23,Z 312.694,A -85,B 0,C 180,E1 -18200.309,E2 -18200.309} C_VEL
LIN {X 0,Y 263.166,Z 312.693,A -85,B 0,C 180,E1 -18205.296,E2 -18205.296} C_VEL
LIN {X 0,Y 263.132,Z 312.71,A -85,B 0,C 180,E1 -18208.735,E2 -18208.735} C_VEL
LIN {X 0,Y 263.122,Z 312.699,A -85,B 0,C 180,E1 -18212.29,E2 -18212.29} C_VEL
LIN {X 0,Y 263.177,Z 312.697,A -85,B 0,C 180,E1 -18216.764,E2 -18216.764} C_VEL
LIN {X 0,Y 263.119,Z 312.707,A -85,B 0,C 180,E1 -18221.595,E2 -18221.595} C_VEL
LIN {X 0,Y 263.119,Z 312.71,A -85,B 0,C 180,E1 -18226.152,E2 -18226.152} C_VEL
LIN {X 0,Y 263.102,Z 312.711,A -85,B 0,C 180,E1 -18230.129,E2 -18230.129} C_VEL
LIN {X 0,Y 263.161,Z 312.693,A -85,B 0,C 180,E1 -18234.02,E2 -18234.02} C_VEL
LIN {X 0,Y 263.13,Z 312.696,A -85,B 0,C 180,E1 -18237.713,E2 -18237.713} C_VEL
LIN {X 0,Y 263.148,Z 312.695,A -85,B 0,C 180,E1 -18238.883,E2 -18238.883} C_VEL
LIN {X 0,Y 264.226,Z 315.659,A -85,B 0,C 180,E1 -18239.13,E2 -18239.13} C_VEL
LIN {X 0,Y 267.134,Z 320.72,A -85,B 0,C 180,E1 -18239.661,E2 -18239.661} C_VEL
LIN {X 0,Y 275.107,Z 336.212,A -85,B 0,C 180,E1 -18241.093,E2 -18241.093} C_VEL
LIN {X 0,Y 279.779,Z 346.675,A -85,B 0,C 180,E1 -18241.925,E2 -18241.925} C_VEL
LIN {X 0,Y 277.77,Z 414.08,A -85,B 0,C 180,E1 -18243.64,E2 -18243.64} C_VEL
LIN {X 0,Y 277.16,Z 426.529,A -85,B 0,C 180,E1 -18244.121,E2 -18244.121} C_VEL
LIN {X 0,Y 276.145,Z 438.868,A -85,B 0,C 180,E1 -18244.87,E2 -18244.87} C_VEL
LIN {X 0,Y 274.798,Z 450.557,A -85,B 0,C 180,E1 -18245.847,E2 -18245.847} C_VEL
LIN {X 0,Y 273.154,Z 461.956,A -85,B 0,C 180,E1 -18247.1,E2 -18247.1} C_VEL
LIN {X 0,Y 271.476,Z 472.22,A -85,B 0,C 180,E1 -18248.553,E2 -18248.553} C_VEL
LIN {X 0,Y 269.839,Z 481.62,A -85,B 0,C 180,E1 -18250.211,E2 -18250.211} C_VEL
LIN {X 0,Y 268.031,Z 490.197,A -85,B 0,C 180,E1 -18252.057,E2 -18252.057} C_VEL
LIN {X 0,Y 266.447,Z 497.27,A -85,B 0,C 180,E1 -18253.923,E2 -18253.923} C_VEL
LIN {X 0,Y 264.93,Z 504.217,A -85,B 0,C 180,E1 -18256.189,E2 -18256.189} C_VEL
LIN {X 0,Y 263.642,Z 509.739,A -85,B 0,C 180,E1 -18258.469,E2 -18258.469} C_VEL
LIN {X 0,Y 262.702,Z 514.062,A -85,B 0,C 180,E1 -18260.765,E2 -18260.765} C_VEL
LIN {X 0,Y 262.156,Z 516.884,A -85,B 0,C 180,E1 -18262.71,E2 -18262.71} C_VEL
LIN {X 0,Y 261.668,Z 519.597,A -85,B 0,C 180,E1 -18265.38,E2 -18265.38} C_VEL
LIN {X 0,Y 261.285,Z 521.202,A -85,B 0,C 180,E1 -18268.46,E2 -18268.46} C_VEL
LIN {X 0,Y 261.257,Z 521.433,A -85,B 0,C 180,E1 -18270.002,E2 -18270.002} C_VEL
LIN {X 0,Y 261.426,Z 520.651,A -85,B 0,C 180,E1 -18273.084,E2 -18273.084} C_VEL
LIN {X 0,Y 261.666,Z 519.683,A -85,B 0,C 180,E1 -18274.623,E2 -18274.623} C_VEL
LIN {X 0,Y 262.143,Z 517.073,A -85,B 0,C 180,E1 -18277.266,E2 -18277.266} C_VEL
LIN {X 0,Y 262.912,Z 512.952,A -85,B 0,C 180,E1 -18280.008,E2 -18280.008} C_VEL
LIN {X 0,Y 263.957,Z 508.298,A -85,B 0,C 180,E1 -18282.3,E2 -18282.3} C_VEL
LIN {X 0,Y 265.32,Z 502.397,A -85,B 0,C 180,E1 -18284.576,E2 -18284.576} C_VEL
LIN {X 0,Y 266.931,Z 495.046,A -85,B 0,C 180,E1 -18286.837,E2 -18286.837} C_VEL
LIN {X 0,Y 268.734,Z 487.501,A -85,B 0,C 180,E1 -18288.686,E2 -18288.686} C_VEL
LIN {X 0,Y 270.625,Z 477.477,A -85,B 0,C 180,E1 -18290.682,E2 -18290.682} C_VEL
LIN {X 0,Y 272.465,Z 466.868,A -85,B 0,C 180,E1 -18292.364,E2 -18292.364} C_VEL
LIN {X 0,Y 274.013,Z 456.808,A -85,B 0,C 180,E1 -18293.627,E2 -18293.627} C_VEL
LIN {X 0,Y 275.502,Z 444.826,A -85,B 0,C 180,E1 -18294.793,E2 -18294.793} C_VEL
LIN {X 0,Y 276.793,Z 431.721,A -85,B 0,C 180,E1 -18295.725,E2 -18295.725} C_VEL
LIN {X 0,Y 277.617,Z 419.566,A -85,B 0,C 180,E1 -18296.298,E2 -18296.298} C_VEL
LIN {X 0,Y 278.86,Z 380.471,A -85,B 0,C 180,E1 -18297.334,E2 -18297.334} C_VEL
LIN {X 0,Y 279.83,Z 346.755,A -85,B 0,C 180,E1 -18298.194,E2 -18298.194} C_VEL
LIN {X 0,Y 271.945,Z 329.82,A -85,B 0,C 180,E1 -18299.6,E2 -18299.6} C_VEL
LIN {X 0,Y 264.493,Z 316.049,A -85,B 0,C 180,E1 -18300.956,E2 -18300.956} C_VEL
LIN {X 0,Y 263.341,Z 313.642,A -85,B 0,C 180,E1 -18301.183,E2 -18301.183} C_VEL
LIN {X 0,Y 263.151,Z 312.706,A -85,B 0,C 180,E1 -18301.281,E2 -18301.281} C_VEL
LIN {X 0,Y 263.178,Z 312.703,A -85,B 0,C 180,E1 -18304.123,E2 -18304.123} C_VEL
LIN {X 0,Y 263.171,Z 312.708,A -85,B 0,C 180,E1 -18307.897,E2 -18307.897} C_VEL
LIN {X 0,Y 263.148,Z 312.71,A -85,B 0,C 180,E1 -18311.89,E2 -18311.89} C_VEL
LIN {X 0,Y 263.134,Z 312.681,A -85,B 0,C 180,E1 -18316.15,E2 -18316.15} C_VEL
LIN {X 0,Y 263.111,Z 312.71,A -85,B 0,C 180,E1 -18320.128,E2 -18320.128} C_VEL
LIN {X 0,Y 263.168,Z 312.697,A -85,B 0,C 180,E1 -18324.019,E2 -18324.019} C_VEL
LIN {X 0,Y 263.138,Z 312.703,A -85,B 0,C 180,E1 -18327.712,E2 -18327.712} C_VEL
LIN {X 0,Y 263.206,Z 312.697,A -85,B 0,C 180,E1 -18331.784,E2 -18331.784} C_VEL
LIN {X 0,Y 263.279,Z 312.681,A -85,B 0,C 180,E1 -18335.252,E2 -18335.252} C_VEL
LIN {X 0,Y 270.497,Z 340.058,A -85,B 0,C 180,E1 -18336.765,E2 -18336.765} C_VEL
LIN {X 0,Y 268.21,Z 397.973,A -85,B 0,C 180,E1 -18339.181,E2 -18339.181} C_VEL
LIN {X 0,Y 267.378,Z 403.719,A -85,B 0,C 180,E1 -18339.405,E2 -18339.405} C_VEL
LIN {X 0,Y 260.969,Z 422.163,A -85,B 0,C 180,E1 -18340.153,E2 -18340.153} C_VEL
LIN {X 0,Y 260.015,Z 427.794,A -85,B 0,C 180,E1 -18340.495,E2 -18340.495} C_VEL
LIN {X 0,Y 259.09,Z 441.66,A -85,B 0,C 180,E1 -18341.594,E2 -18341.594} C_VEL
LIN {X 0,Y 258.242,Z 454.885,A -85,B 0,C 180,E1 -18342.989,E2 -18342.989} C_VEL
LIN {X 0,Y 257.451,Z 465.214,A -85,B 0,C 180,E1 -18344.361,E2 -18344.361} C_VEL
LIN {X 0,Y 256.49,Z 477.183,A -85,B 0,C 180,E1 -18346.33,E2 -18346.33} C_VEL
LIN {X 0,Y 255.797,Z 486.048,A -85,B 0,C 180,E1 -18348.108,E2 -18348.108} C_VEL
LIN {X 0,Y 255.084,Z 495.718,A -85,B 0,C 180,E1 -18350.485,E2 -18350.485} C_VEL
LIN {X 0,Y 254.578,Z 503.52,A -85,B 0,C 180,E1 -18352.864,E2 -18352.864} C_VEL
LIN {X 0,Y 254.274,Z 509.783,A -85,B 0,C 180,E1 -18355.244,E2 -18355.244} C_VEL
LIN {X 0,Y 254.211,Z 514.73,A -85,B 0,C 180,E1 -18357.623,E2 -18357.623} C_VEL
LIN {X 0,Y 254.144,Z 518.503,A -85,B 0,C 180,E1 -18360,E2 -18360} C_VEL
LIN {X 0,Y 254.261,Z 520.425,A -85,B 0,C 180,E1 -18361.584,E2 -18361.584} C_VEL
LIN {X 0,Y 254.493,Z 521.929,A -85,B 0,C 180,E1 -18363.166,E2 -18363.166} C_VEL
LIN {X 0,Y 254.784,Z 523.018,A -85,B 0,C 180,E1 -18364.747,E2 -18364.747} C_VEL
LIN {X 0,Y 255.133,Z 523.662,A -85,B 0,C 180,E1 -18366.326,E2 -18366.326} C_VEL
LIN {X 0,Y 256.466,Z 523.742,A -85,B 0,C 180,E1 -18369.463,E2 -18369.463} C_VEL
LIN {X 0,Y 257.461,Z 523.18,A -85,B 0,C 180,E1 -18371.016,E2 -18371.016} C_VEL
LIN {X 0,Y 258.478,Z 522.199,A -85,B 0,C 180,E1 -18372.563,E2 -18372.563} C_VEL
LIN {X 0,Y 259.614,Z 520.812,A -85,B 0,C 180,E1 -18374.101,E2 -18374.101} C_VEL
LIN {X 0,Y 261.96,Z 517.912,A -85,B 0,C 180,E1 -18376.362,E2 -18376.362} C_VEL
LIN {X 0,Y 264.554,Z 514.028,A -85,B 0,C 180,E1 -18378.59,E2 -18378.59} C_VEL
LIN {X 0,Y 267.579,Z 509.044,A -85,B 0,C 180,E1 -18380.768,E2 -18380.768} C_VEL
LIN {X 0,Y 271.638,Z 501.702,A -85,B 0,C 180,E1 -18383.238,E2 -18383.238} C_VEL
LIN {X 0,Y 275.627,Z 493.781,A -85,B 0,C 180,E1 -18385.283,E2 -18385.283} C_VEL
LIN {X 0,Y 279.969,Z 484.144,A -85,B 0,C 180,E1 -18387.266,E2 -18387.266} C_VEL
LIN {X 0,Y 284.219,Z 473.369,A -85,B 0,C 180,E1 -18389.031,E2 -18389.031} C_VEL
LIN {X 0,Y 288.445,Z 461.297,A -85,B 0,C 180,E1 -18390.572,E2 -18390.572} C_VEL
LIN {X 0,Y 292.425,Z 447.655,A -85,B 0,C 180,E1 -18391.92,E2 -18391.92} C_VEL
LIN {X 0,Y 295.475,Z 434.964,A -85,B 0,C 180,E1 -18392.861,E2 -18392.861} C_VEL
LIN {X 0,Y 298.084,Z 421.38,A -85,B 0,C 180,E1 -18393.609,E2 -18393.609} C_VEL
LIN {X 0,Y 304.816,Z 382.738,A -85,B 0,C 180,E1 -18395.35,E2 -18395.35} C_VEL
LIN {X 0,Y 302.744,Z 378.491,A -85,B 0,C 180,E1 -18397.023,E2 -18397.023} C_VEL
LIN {X 0,Y 301.566,Z 376.344,A -85,B 0,C 180,E1 -18398.148,E2 -18398.148} C_VEL
LIN {X 0,Y 300.143,Z 373.91,A -85,B 0,C 180,E1 -18399.833,E2 -18399.833} C_VEL
LIN {X 0,Y 298.524,Z 371.894,A -85,B 0,C 180,E1 -18403.127,E2 -18403.127} C_VEL
LIN {X 0,Y 298.312,Z 372.401,A -85,B 0,C 180,E1 -18405.535,E2 -18405.535} C_VEL
LIN {X 0,Y 298.549,Z 373.866,A -85,B 0,C 180,E1 -18407.064,E2 -18407.064} C_VEL
LIN {X 0,Y 300.191,Z 378.741,A -85,B 0,C 180,E1 -18410.244,E2 -18410.244} C_VEL
LIN {X 0,Y 301.883,Z 384.35,A -85,B 0,C 180,E1 -18412.33,E2 -18412.33} C_VEL
LIN {X 0,Y 303.367,Z 389.463,A -85,B 0,C 180,E1 -18413.776,E2 -18413.776} C_VEL
LIN {X 0,Y 303.193,Z 395.631,A -85,B 0,C 180,E1 -18414.458,E2 -18414.458} C_VEL
LIN {X 0,Y 295.316,Z 441.105,A -85,B 0,C 180,E1 -18416.506,E2 -18416.506} C_VEL
LIN {X 0,Y 291.969,Z 455.282,A -85,B 0,C 180,E1 -18417.35,E2 -18417.35} C_VEL
LIN {X 0,Y 287.688,Z 469.882,A -85,B 0,C 180,E1 -18418.52,E2 -18418.52} C_VEL
LIN {X 0,Y 283.341,Z 482.446,A -85,B 0,C 180,E1 -18419.847,E2 -18419.847} C_VEL
LIN {X 0,Y 278.965,Z 493.83,A -85,B 0,C 180,E1 -18421.4,E2 -18421.4} C_VEL
LIN {X 0,Y 274.926,Z 503.352,A -85,B 0,C 180,E1 -18423.014,E2 -18423.014} C_VEL
LIN {X 0,Y 270.645,Z 512.886,A -85,B 0,C 180,E1 -18425.039,E2 -18425.039} C_VEL
LIN {X 0,Y 266.701,Z 521.022,A -85,B 0,C 180,E1 -18427.218,E2 -18427.218} C_VEL
LIN {X 0,Y 262.934,Z 528.235,A -85,B 0,C 180,E1 -18429.665,E2 -18429.665} C_VEL
LIN {X 0,Y 260.431,Z 533.346,A -85,B 0,C 180,E1 -18431.919,E2 -18431.919} C_VEL
LIN {X 0,Y 258.148,Z 537.442,A -85,B 0,C 180,E1 -18434.2,E2 -18434.2} C_VEL
LIN {X 0,Y 256.907,Z 539.633,A -85,B 0,C 180,E1 -18435.745,E2 -18435.745} C_VEL
LIN {X 0,Y 255.973,Z 541.409,A -85,B 0,C 180,E1 -18437.31,E2 -18437.31} C_VEL
LIN {X 0,Y 255.232,Z 542.757,A -85,B 0,C 180,E1 -18438.885,E2 -18438.885} C_VEL
LIN {X 0,Y 254.295,Z 544.252,A -85,B 0,C 180,E1 -18442.056,E2 -18442.056} C_VEL
LIN {X 0,Y 254.086,Z 544.281,A -85,B 0,C 180,E1 -18444.721,E2 -18444.721} C_VEL
LIN {X 0,Y 254.15,Z 543.618,A -85,B 0,C 180,E1 -18446.828,E2 -18446.828} C_VEL
LIN {X 0,Y 254.17,Z 544.24,A -85,B 0,C 180,E1 -18448.414,E2 -18448.414} C_VEL
LIN {X 0,Y 254.308,Z 544.464,A -85,B 0,C 180,E1 -18449.998,E2 -18449.998} C_VEL
LIN {X 0,Y 254.219,Z 544.233,A -85,B 0,C 180,E1 -18451.583,E2 -18451.583} C_VEL
LIN {X 0,Y 254.131,Z 543.602,A -85,B 0,C 180,E1 -18453.169,E2 -18453.169} C_VEL
LIN {X 0,Y 254.046,Z 542.232,A -85,B 0,C 180,E1 -18455.179,E2 -18455.179} C_VEL
LIN {X 0,Y 254.262,Z 539.21,A -85,B 0,C 180,E1 -18457.942,E2 -18457.942} C_VEL
LIN {X 0,Y 254.688,Z 535.503,A -85,B 0,C 180,E1 -18460.331,E2 -18460.331} C_VEL
LIN {X 0,Y 255.437,Z 530.658,A -85,B 0,C 180,E1 -18462.714,E2 -18462.714} C_VEL
LIN {X 0,Y 256.809,Z 524.546,A -85,B 0,C 180,E1 -18465.067,E2 -18465.067} C_VEL
LIN {X 0,Y 258.451,Z 516.935,A -85,B 0,C 180,E1 -18467.403,E2 -18467.403} C_VEL
LIN {X 0,Y 260.001,Z 509.122,A -85,B 0,C 180,E1 -18469.335,E2 -18469.335} C_VEL
LIN {X 0,Y 261.949,Z 499.576,A -85,B 0,C 180,E1 -18471.234,E2 -18471.234} C_VEL
LIN {X 0,Y 264.081,Z 488.991,A -85,B 0,C 180,E1 -18472.904,E2 -18472.904} C_VEL
LIN {X 0,Y 265.853,Z 478.747,A -85,B 0,C 180,E1 -18474.188,E2 -18474.188} C_VEL
LIN {X 0,Y 267.48,Z 467.578,A -85,B 0,C 180,E1 -18475.273,E2 -18475.273} C_VEL
LIN {X 0,Y 269.046,Z 454.343,A -85,B 0,C 180,E1 -18476.206,E2 -18476.206} C_VEL
LIN {X 0,Y 270.133,Z 441.431,A -85,B 0,C 180,E1 -18476.802,E2 -18476.802} C_VEL
LIN {X 0,Y 271.883,Z 384.051,A -85,B 0,C 180,E1 -18478.323,E2 -18478.323} C_VEL
LIN {X 0,Y 268.276,Z 354.701,A -85,B 0,C 180,E1 -18479.611,E2 -18479.611} C_VEL
LIN {X 0,Y 266.42,Z 342.033,A -85,B 0,C 180,E1 -18480.22,E2 -18480.22} C_VEL
LIN {X 0,Y 259.304,Z 322.595,A -85,B 0,C 180,E1 -18481.747,E2 -18481.747} C_VEL
LIN {X 0,Y 256.193,Z 313.572,A -85,B 0,C 180,E1 -18482.603,E2 -18482.603} C_VEL
LIN {X 0,Y 256.118,Z 313.577,A -85,B 0,C 180,E1 -18487.271,E2 -18487.271} C_VEL
LIN {X 0,Y 256.05,Z 313.587,A -85,B 0,C 180,E1 -18491.202,E2 -18491.202} C_VEL
LIN {X 0,Y 256.032,Z 313.591,A -85,B 0,C 180,E1 -18495.534,E2 -18495.534} C_VEL
LIN {X 0,Y 256.003,Z 313.592,A -85,B 0,C 180,E1 -18498.786,E2 -18498.786} C_VEL
LIN {X 0,Y 256.092,Z 313.581,A -85,B 0,C 180,E1 -18502.861,E2 -18502.861} C_VEL
LIN {X 0,Y 256.058,Z 313.586,A -85,B 0,C 180,E1 -18506.706,E2 -18506.706} C_VEL
LIN {X 0,Y 256.033,Z 313.589,A -85,B 0,C 180,E1 -18510.39,E2 -18510.39} C_VEL
LIN {X 0,Y 256.061,Z 313.582,A -85,B 0,C 180,E1 -18513.951,E2 -18513.951} C_VEL
LIN {X 0,Y 256.055,Z 313.591,A -85,B 0,C 180,E1 -18517.402,E2 -18517.402} C_VEL
LIN {X 0,Y 256.121,Z 313.564,A -85,B 0,C 180,E1 -18520.775,E2 -18520.775} C_VEL
LIN {X 0,Y 256.222,Z 313.548,A -85,B 0,C 180,E1 -18524.08,E2 -18524.08} C_VEL
LIN {X 0,Y 256.279,Z 313.56,A -85,B 0,C 180,E1 -18527.327,E2 -18527.327} C_VEL
LIN {X 0,Y 256.426,Z 313.537,A -85,B 0,C 180,E1 -18530.622,E2 -18530.622} C_VEL
LIN {X 0,Y 256.445,Z 313.505,A -85,B 0,C 180,E1 -18533.707,E2 -18533.707} C_VEL
LIN {X 0,Y 256.688,Z 313.504,A -85,B 0,C 180,E1 -18538.431,E2 -18538.431} C_VEL
LIN {X 0,Y 256.69,Z 313.506,A -85,B 0,C 180,E1 -18541.569,E2 -18541.569} C_VEL
LIN {X 0,Y 256.43,Z 313.538,A -85,B 0,C 180,E1 -18546.681,E2 -18546.681} C_VEL
LIN {X 0,Y 256.419,Z 313.536,A -85,B 0,C 180,E1 -18549.465,E2 -18549.465} C_VEL
LIN {X 0,Y 256.224,Z 313.567,A -85,B 0,C 180,E1 -18554.292,E2 -18554.292} C_VEL
LIN {X 0,Y 256.166,Z 313.562,A -85,B 0,C 180,E1 -18557.565,E2 -18557.565} C_VEL
LIN {X 0,Y 256.135,Z 313.58,A -85,B 0,C 180,E1 -18561.111,E2 -18561.111} C_VEL
LIN {X 0,Y 256.152,Z 313.565,A -85,B 0,C 180,E1 -18565.125,E2 -18565.125} C_VEL
LIN {X 0,Y 256.05,Z 313.588,A -85,B 0,C 180,E1 -18569.608,E2 -18569.608} C_VEL
LIN {X 0,Y 256.06,Z 313.585,A -85,B 0,C 180,E1 -18573.294,E2 -18573.294} C_VEL
LIN {X 0,Y 256.109,Z 313.574,A -85,B 0,C 180,E1 -18577.272,E2 -18577.272} C_VEL
LIN {X 0,Y 256.049,Z 313.588,A -85,B 0,C 180,E1 -18581.205,E2 -18581.205} C_VEL
LIN {X 0,Y 256.049,Z 313.59,A -85,B 0,C 180,E1 -18585.532,E2 -18585.532} C_VEL
LIN {X 0,Y 256.051,Z 313.591,A -85,B 0,C 180,E1 -18588.798,E2 -18588.798} C_VEL
LIN {X 0,Y 256.129,Z 313.56,A -85,B 0,C 180,E1 -18592.869,E2 -18592.869} C_VEL
LIN {X 0,Y 256.073,Z 313.583,A -85,B 0,C 180,E1 -18596.71,E2 -18596.71} C_VEL
LIN {X 0,Y 256.104,Z 313.687,A -85,B 0,C 180,E1 -18597.964,E2 -18597.964} C_VEL
LIN {X 0,Y 257.131,Z 316.485,A -85,B 0,C 180,E1 -18598.198,E2 -18598.198} C_VEL
LIN {X 0,Y 258.476,Z 318.746,A -85,B 0,C 180,E1 -18598.457,E2 -18598.457} C_VEL
LIN {X 0,Y 266.3,Z 333.107,A -85,B 0,C 180,E1 -18599.936,E2 -18599.936} C_VEL
LIN {X 0,Y 273.5,Z 348.559,A -85,B 0,C 180,E1 -18601.27,E2 -18601.27} C_VEL
LIN {X 0,Y 271.258,Z 419.014,A -85,B 0,C 180,E1 -18603.134,E2 -18603.134} C_VEL
LIN {X 0,Y 270.394,Z 431.739,A -85,B 0,C 180,E1 -18603.73,E2 -18603.73} C_VEL
